(* CoDeSys 2.3 export: BPROOpcion2.EXP *)
(* Libraries: STANDARD.LIB 5.6.98 11:03:02, TcBase.lib 14.5.09 11:14:08, TcBaseMath.lib 27.7.04 11:07:56, TcDrive.lib 25.1.17 09:42:28, TcEtherCAT.lib 30.11.16 19:52:18, TcMath.lib 23.9.04 15:15:30, TcMC2.lib 13.9.17 10:18:38, TcMc2Drive.lib 9.10.17 15:27:28, TcNC.lib 10.10.08 17:55:34, TcSystem.lib 7.6.16 11:01:22, TcTestAndSet.lib 23.2.09 11:50:08, TcUtilities.lib 3.2.16 16:08:58 *)

(* Task configuration *)
TASK Standard (PRIORITY := 0, INTERVAL := T#10ms);
MAIN
END_TASK

(* Global variable list: Global_Variables *)
VAR_GLOBAL
	sCurrentProgram : STRING(20) := 'None';			(* Current Program Loaded or Saved *)

	(* ***** SECURITY ***** *)
	sUsername: STRING := '';
	sPassword : STRING := '';
	sSavePassword : STRING := '';					(* Password Variable for the Save Screen *)
	OldUserLevel : INT := 0;						(* Previous User Level before logging in *)
	CurrentUserLevel : INT :=0;						(* Current User Level*)
	bWrongPassword :BOOL:=FALSE;				(*The password is not correct*)
	bWrongSavePassword :BOOL:=FALSE;				(*The password is not correct*)
	bUserNameHandshake: BOOL := FALSE;			(* Handshake bit to tell panels the User Name Input was received *)
	bPasswordHandshake: BOOL := FALSE;			(* Handshake bit to tell panels the Password Input was received *)
	bSavePasswordHandshake: BOOL := FALSE;		(* Handshake bit to tell panels the Password Input was received *)
	(* SECURITY LEVELS *)
	(* Level 7 - Kays is no longer needed *)
	sUsernameKays : STRING := 'Kays';					(* Username for Kays Engineering *)
	sUsernameKaysLC : STRING := 'kaysengineering';		(* Username for Kays Engineering - Lower Case*)
	sUsernameKaysEngineering : STRING := 'KaysEngineering';		(* Username for Kays Engineering *)
	sPasswordKays : STRING := 'Dehoff';					(* Password for Kays Engineering - Ed's Birthday *)
	(* Level 6 - Maintenance *)
	sUsernameMaint : STRING := 'Maint';					(* Username for Maint *)
	sUsernameMaintLC : STRING := 'maint';				(* Username for maint *)
	sUsernameMaintenance : STRING := 'Maintenance';	(* Username for Maintenance *)
	sUsernameMaintenanceLC : STRING := 'maintenance';	(* Username for maintenance - Lower Case *)
	sPasswordMaint : STRING := 'lazarini';					(* Password for Maintenance - Toggling on the keyboard with the numbers*)
	sPasswordMaintenance : STRING := 'LAZARINI';		(* Password for Maintenance - Toggling on the keyboard with the numbers*)
	(* Level 5 - Supervisor *)
	sUsernameSuper : STRING := 'Super';				(* Username for Super *)
	sUsernameSuperLC : STRING := 'super';				(* Username for super *)
	sUsernameSupervisor : STRING := 'Supervisor';		(* Username for Supervisor *)
	sUsernameSupervisorLC : STRING := 'supervisor';		(* Username for Supervisor  - Lower Case*)
	sPasswordSupervisorUC : STRING := 'ROYALS';		(* Password for Supervisor - Start at 1 and go down then start at 2 and go down keyboard *)
	sPasswordSupervisor : STRING := 'royals';			(* Password for Supervisor - Start at 1 and go down then start at 2 and go down keyboard  - Lower Case*)
	sPasswordSuperUC : STRING := 'ROYALS';		(* Password for Supervisor - Start at 1 and go down then start at 2 and go down keyboard *)
	sPasswordSuper : STRING := 'royals';			(* Password for Supervisor - Start at 1 and go down then start at 2 and go down keyboard  - Lower Case*)

	(* Faulting Variables *)
	bMachineFault: BOOL := FALSE; 					(* Machine Fault Indicator *)
	bMachineWarning: BOOL := FALSE; 				(* Machine Warning Indicator *)
	nFaultArrayIndex : UDINT := 1;
	nWarningArrayIndex : UDINT := 1;
	nModeError : ModeErrors := Er_NoModeError;		(* Errors for different functions *)
	bCoolantTempWarning : BOOL := FALSE;
	bCoolantTempFault : BOOL := FALSE;
	fbCommonFautlResetTON: TON;				(* Trigger of Common Button to Reset Faults *)
	bAFaultResetInternal : BOOL := FALSE;			(* Side A Internal Fault Reset. Triggered by VFD's Ready *)
	bBFaultResetInternal : BOOL := FALSE;			(* Side B Internal Fault Reset. Triggered by VFD's Ready *)
	nActiveFaults: ARRAY[1..4] OF DWORD := 4(0);
	nActiveWarnings: ARRAY[1..4] OF DWORD := 4(0);
	nFaultState: UDINT := 0;
	arrFaultHistory : ARRAY[1..80] OF STRING (52) := 80(''); (* Fault History array *)
	(* Helper Bits *)
	nSetupErrorID: INT :=0;							(* Setup Mode Error Occurred *)
	bLoadSideNotSelected : BOOL := FALSE;
	bTransferError: BOOL := FALSE;					(* An Error Occurred with the Transfer Cycle *)
	nTransferErrorID: INT := 0;						(* Transfer Error ID *)
	sTransferErrorText : STRING := '';				(* Transfer Error Text *)
	(* Parts Tracking *)
	bSideADrilledParts: BOOL := FALSE;				(* Tracking Bit - Side A Completed Drilled parts *)
	bSideBDrilledParts: BOOL := FALSE;				(* Tracking Bit - Side B Completed Drilled parts *)
	fbCoolantLevelDelayTOF: TOF;					(* Delay of the Lowe level switch *)

	(* Status Variables *)
	bMachineMode: BOOL := FALSE;				(* FALSE-->Manual, TRUE-->Automatic *)
	bSetup: BOOL := FALSE;						(* At least one Side in Setup Mode *)
	bSetupA: BOOL := FALSE;						(* In Setup Mode Side A *)
	bSetupB: BOOL := FALSE;						(* In Setup Mode Side B*)
	bInCycle: BOOL := FALSE;						(* In Cycle Flag *)

	(* Cycle Variables *)
	nCycleTimeMinutes : UDINT := 0;
	nCycleTimeSeconds : UDINT := 0;
	nAutoModeState: AutoModeStates := AM_NotInCycle;	(* Counter for Auto Mode State *)
	nAutoCycleStep : AutoCycleStates := AC_Init;		(* Counter for Auto Cycle State *)
	nAC_UnclampStep: INT := 0;					(* Counter for the AC Unclamp Step*)
	bUnloadSideClearOfParts: BOOL :=FALSE;		(* All Unload Side Proxes are off *)
	nCellRunoutCounter: UINT:=0;					(* Counter to keep track of transfer cycles durring Cell Runout *)

	bAutoClampAStart: BOOL := FALSE;				(* Automatic cycle Side A Clamp Parts Tailstock Input *)
	bAutoClampADone: BOOL := FALSE;				(* Automatic cycle Side A Clamp Parts Tailstock Done Output *)
	bAutoClampBStart: BOOL := FALSE;				(* Automatic cycle Side B Clamp PartsTailstock Input *)
	bAutoClampBDone: BOOL := FALSE;				(* Automatic cycle Side B Clamp Parts Tailstock Done Output *)
	bAutoUnclampAStart: BOOL := FALSE;			(* Automatic Side A Unclamp Parts Tailstock Input *)
	bAutoUnclampADone: BOOL := FALSE;			(* Automatic cycle Side A Unclamp Parts Tailstock Done Output *)
	bAutoUnclampBStart: BOOL := FALSE;			(* Automatic Side B Unclamp Parts Tailstock Input *)
	bAutoUnclampBDone: BOOL := FALSE;			(* Automatic cycle Side B Unclamp Parts Tailstock Done Output *)
	bLoadPartsConfirmed: BOOL := FALSE;			(* Operator Confirmed Load Parts In Cycle *)
	bUnloadPartsConfirmed: BOOL := FALSE;			(* Operator Confirmed Unload Parts In Cycle *)
	bAutoTransferPartsToDrill: BOOL := FALSE;		(*Auto Trigger the Transfer to Raise and move parts to Drill Postion*)
	bAutoTransferDownAndLoad : BOOL := FALSE;	(*Auto Trigger the Transfer to lower and move Load Postion*)
	fbProx516TON: TON;							(* Delay of the Transfer Carriage Up Prox *)
	fbProx517TON: TON;							(* Delay of the Transfer Carriage Down Prox *)
	bAutoUpDelayWhileUnclamp: BOOL := FALSE;	(* Auto Helper bit to turn off the up Solenoid when the Unclamp is firing*)

	(*	SERVO VARIABLES *)
	bMCResetRequest: BOOL := FALSE;				(* Request a reset of the NC Axis *)
	bZWADriveResetRequest : BOOL := FALSE;		(* A Side ZW Drive Reset Request *)
	bZBDriveResetRequest : BOOL := FALSE;			(* B Side ZW Drive Reset Request *)
	bZWBDriveResetRequest : BOOL := FALSE;		(* B Side ZW Drive Reset Request *)
	bUDriveResetRequest : BOOL := FALSE;			(* U Axis Drive Reset Request *)
	DriveZAWAdinputs AT %I*: INT;

(* ZA AXIS *)
	stZAAxis: AXIS_REF;
	nZAAxisDiagNumber AT %I*: UDINT := 0;
	nServoZAThrust AT %I* : INT :=0;
	fbZAAxisStop: MC_Stop;
	bZAStop: BOOL := FALSE;
	bZAMCResetRequest: BOOL := FALSE;			(* Request a reset of the NC Axis *)
	fbZAAxisMCReset: MC_Reset;
	fbZAAxisDriveReset : FB_SoEReset;

	bZAAxisEnable: BOOL;
	fbZAAxisPower: MC_Power;
	fbZAAxisMove: MC_MoveAbsolute;
	fbZAAxisSetZero: MC_Home;
	bZAAxisPower: BOOL := FALSE;
	bZAAxisHome: BOOL := FALSE;
	bZAAxisMove: BOOL := FALSE;
	bZAAxisSetZero: BOOL := FALSE;
	fZAMoveVelocity : LREAL := 25.0;
	fZAMovePosition : LREAL := 0.0;
	bZADeCtrlEnable: BOOL := FALSE;				(* Enable for the FB to move off of the Overtravel *)

(* WA AXIS*)
	stWAAxis: AXIS_REF;							(* A Side Tailstock Axis cyclic Interface *)
	nWAAxisDiagNumber AT %I*: UDINT := 0;
	nWAAxisThrust AT %I* : INT :=0;
	fbWAAxisStop: MC_Stop;
	bWAStop: BOOL := FALSE;
	bWAMCResetRequest: BOOL := FALSE;			(* Request a reset of the WA NC Axis *)
	fbWAAxisMCReset: MC_Reset;
	fbWAAxisDriveReset : FB_SoEReset;
	nWATorqeLimitValue AT %Q* : INT := 1000;
	fbWAAxisHome: MC_Home;
	bWAAxisHome: BOOL := FALSE;					(*Trigger the home of WA while homing Automation*)

	DriveZBWBdinputs AT %I*: INT;
(* ZB AXIS *)
	stZBAxis: AXIS_REF;
	nZBAxisDiagNumber AT %I*: UDINT := 0;
	nServoZBThrust AT %I* : INT :=0;
	fbZBAxisStop: MC_Stop;
	bZBStop: BOOL := FALSE;
	bZBMCResetRequest: BOOL := FALSE;			(* Request a reset of the ZA NC Axis *)
	fbZBAxisMCReset: MC_Reset;
	fbZBAxisDriveReset : FB_SoEReset;

	bZBAxisEnable: BOOL;
	fbZBAxisPower: MC_Power;
	fbZBAxisMove: MC_MoveAbsolute;
	fbZBAxisSetZero: MC_Home;
	bZBAxisPower: BOOL := FALSE;
	bZBAxisMove: BOOL := FALSE;
	bZBAxisSetZero: BOOL := FALSE;
	fZBMoveVelocity : LREAL := 25.0;
	fZBMovePosition : LREAL := 0.0;
	bZBDeCtrlEnable: BOOL := FALSE;				(* Enable for the FB to move off of the Overtravel *)

(* WB AXIS *)
	stWBAxis: AXIS_REF;							(* Transfer Axis cyclic Interface *)
	nWBAxisDiagNumber AT %I*: UDINT := 0;
	nWBAxisThrust AT %I* : INT :=0;
	fbWBAxisStop: MC_Stop;
	bWBStop: BOOL := FALSE;
	bWBMCResetRequest: BOOL := FALSE;			(* Request a reset of theWB  NC Axis *)
	fbWBAxisMCReset : MC_Reset;
	fbWBAxisDriveReset : FB_SoEReset;
	nWBTorqeLimitValue AT %Q* : INT  := 1000;
	fbHomeWB: MC_Home;
	bWBAxisHome: BOOL := FALSE;					(*Trigger the home of WB while homing Automation*)

	DriveUdinputs AT %I*: INT;
(* U AXIS 		Also Called X Axis on Screens *)
	stUAxis: AXIS_REF;							(* Transfer Axis cyclic Interface *)
	nUAxisDiagNumber AT %I*: UDINT := 0;
	nUAxisThrust AT %I* : INT :=0;
	fbUAxisStop: MC_Stop;
	bUStop: BOOL := FALSE;
	bUMCResetRequest: BOOL := FALSE;			(* Request a reset of the U NC Axis *)
	fbUAxisMCReset : MC_Reset;
	fbUAxisDriveReset : FB_SoEReset;
	fbTransferAxisHome: MC_Home;
	bUAxisHome: BOOL := FALSE;					(*Trigger the home of U Axis while homing Automation*)
	fTransferMoveVelo : LREAL := 0.0;				(* Velocity to pass to the U Axis Move FB *)

(* MPG Axis Definitions *)
	stAxisMPG_A : Axis_REF;						(* Side A MPG Axis Cyclic Interface *)
	fbMPGAAxisMCReset: MC_Reset;
	stAxisMPG_B : Axis_REF;						(* Side A MPG Axis Cyclic Interface *)
	fbMPGBAxisMCReset: MC_Reset;
	bMPGA_MCResetRequest: BOOL := FALSE;		(* Axis Reset of the MPGA Axis *)
	bMPGB_MCResetRequest: BOOL := FALSE;		(* Axis Reset of the MPGB Axis *)
	bMPGAOn: BOOL := FALSE;						(* MPG A has an axis selected *)
	bMPGBOn: BOOL := FALSE;						(* MPG B has an axis selected *)

(* VFD Control Variables - EtherCAT Emerson *)
	fbGetAMS: FB_GetAxisAmsAddr;
	fbVFD_A1: FB_EtherCAT_Emerson;
	bVFD_A1DataValid AT %I*: BOOL;				(* Must Asign to VFD WcStateIn in System Manager*)
	fbVFD_A2: FB_EtherCAT_Emerson;
	bVFD_A2DataValid AT %I*: BOOL;				(* Must Asign to VFD WcStateIn in System Manager*)
	fbVFD_A3: FB_EtherCAT_Emerson;
	bVFD_A3DataValid AT %I*: BOOL;				(* Must Asign to VFD WcStateIn in System Manager*)
	fbVFD_B1: FB_EtherCAT_Emerson;
	bVFD_B1DataValid AT %I*: BOOL;				(* Must Asign to VFD WcStateIn in System Manager*)
	fbVFD_B2: FB_EtherCAT_Emerson;
	bVFD_B2DataValid AT %I*: BOOL;				(* Must Asign to VFD WcStateIn in System Manager*)
	fbVFD_B3: FB_EtherCAT_Emerson;
	bVFD_B3DataValid AT %I*: BOOL;				(* Must Asign to VFD WcStateIn in System Manager*)
	bVFD_ARun: BOOL := FALSE;
	bVFD_BRun: BOOL := FALSE;
	bVFDControlDirection: BOOL := FALSE;
	fVFDControlRatio: LREAL := 1.0;
	bVFD_A1UpToSpeed: BOOL := FALSE;
	bVFD_A1Error: BOOL := FALSE;
	nVFD_A1ErrorID: UDINT := 0;
	stVFD_A1DriveInfo: Ke_VFDInfo;
	bVFD_A2UpToSpeed: BOOL := FALSE;
	bVFD_A2Error: BOOL := FALSE;
	nVFD_A2ErrorID: UDINT := 0;
	stVFD_A2DriveInfo: Ke_VFDInfo;
	bVFD_A3UpToSpeed: BOOL := FALSE;
	bVFD_A3Error: BOOL := FALSE;
	nVFD_A3ErrorID: UDINT := 0;
	stVFD_A3DriveInfo: Ke_VFDInfo;
	bVFD_B1UpToSpeed: BOOL := FALSE;
	bVFD_B1Error: BOOL := FALSE;
	nVFD_B1ErrorID: UDINT := 0;
	stVFD_B1DriveInfo: Ke_VFDInfo;
	bVFD_B2UpToSpeed: BOOL := FALSE;
	bVFD_B2Error: BOOL := FALSE;
	nVFD_B2ErrorID: UDINT := 0;
	stVFD_B2DriveInfo: Ke_VFDInfo;
	bVFD_B3UpToSpeed: BOOL := FALSE;
	bVFD_B3Error: BOOL := FALSE;
	nVFD_B3ErrorID: UDINT := 0;
	stVFD_B3DriveInfo: Ke_VFDInfo;
	nVFD_A1Addr AT %I*: UINT := 0;						(*Spindle#A1 VFD Slave Addres Input Variable*)
	nVFD_A2Addr AT %I*: UINT := 0;						(*Spindle#A1 VFD Slave Addres Input Variable*)
	nVFD_A3Addr AT %I*: UINT := 0;						(*Spindle#A1 VFD Slave Addres Input Variable*)
	nVFD_B1Addr AT %I*: UINT := 0;						(*Spindle#A1 VFD Slave Addres Input Variable*)
	nVFD_B2Addr AT %I*: UINT := 0;						(*Spindle#A1 VFD Slave Addres Input Variable*)
	nVFD_B3Addr AT %I*: UINT := 0;						(*Spindle#A1 VFD Slave Addres Input Variable*)


(* Solenoid Auto Control Variables *)
	bAutoLower: BOOL := FALSE;						(* Auto Lower Transfer Carrier Cylinder*)
	bAutoRaise: BOOL := FALSE;						(* Auto Raise Transfer Carrier Cylinder*)
	bAAutoOpenCollet: BOOL := FALSE;					(* Auto Control to Open the Collets on Side A*)
	bAAutoCloseCollet: BOOL := FALSE;					(* Auto Control to Close the Collets on Side A*)
	bBAutoOpenCollet: BOOL := FALSE;					(* Auto Control to Open the Collets on Side B*)
	bBAutoCloseCollet: BOOL := FALSE;					(* Auto Control to Close the Collets on Side B*)
	bAAutoEjectorsAdvance: BOOL := FALSE;				(* Auto Control to Advance the Ejectors on Side A *)
	bAAutoEjectorsRetract: BOOL := FALSE;				(* Auto Control to Retract the Ejectors on Side A *)
	bBAutoEjectorsAdvance: BOOL := FALSE;				(* Auto Control to Advance the Ejectors on Side A *)
	bBAutoEjectorsRetract: BOOL := FALSE;				(* Auto Control to Retract the Ejectors on Side A *)

	bWandUAxisHomed: BOOL := FALSE;				(* The W and U Axis are Homed*)

	nAEjectorAdvancedState: USINT := 0;
	nAEjectorRetractedState: USINT := 0;
	nBEjectorAdvancedState: USINT := 0;
	nBEjectorRetractedState: USINT := 0;

(* Tailstock Variables *)
	Side_A_Fixture: FB_FixtureControl;					(*Side A Tailstock Control FB*)
	Side_B_Fixture: FB_FixtureControl;					(*Side B Tailstock Control FB*)
	fWAxisFastVelocity: LREAL := 0.0;					(*WA and WB Axis Velocity to Feed to Tailstock FB*)
	fWAxisClampVelocity: LREAL := 0.0;					(*WA and WB Axis Clamp Velocity to Feed to Tailstock FB*)

END_VAR

VAR_GLOBAL PERSISTENT

	sSerialNumber : STRING(20) := 'DH-2062';				(* This holds the serial number of the machine *)
	sKaysJobNumber  : STRING(20) := '6216';				(* This holds the Kayse Engineering Job number of the machine *)
	sModelNumber : STRING(20) := '6-Spindle Special';		(* This variable holds the model of the machine *)
	sCustomerName : STRING(20) := 'ARBOMEX';			(* This variable holds the customers name *)
	nMachineNumber : UDINT := 7;						(* The Machine Number designates what number the machines were delivered in for this series of special machines *)
	sProductionDate : STRING(10) := '01/2016';			(* This variable holds the date of production and should match that of the machine tags *)

	sLoadSideSet : STRING(30) :='None';					(* Holds the side that is currently set as Infeed *)
	bSideAEnabled : BOOL := TRUE;					(* Enable of Machine Side A *)
	bSideBEnabled : BOOL := TRUE;					(* Enable of Machine Side B *)
	fFlowMonitorMax : LREAL := 0;						(* Max set in program *)

	nMaxCycles : UDINT := 0;							(* Max Cycles set in program *)
	nCyclesComplete : UDINT := 0;						(* Completed # of Cycles since Reset *)

	sLastLoadedPartProgramName : STRING(25) := 'None';	(* Stores the Name of the Last Part Program Loaded *)
	nMotorNominalRPM : UDINT := 3460;

	(* Tailstock Variables *)
	nWAAxisThrustMax: UDINT := 40;					(* Tailstock WA Axis Max Thrust *)
	nWBAxisThrustMax: UDINT := 40;					(* Tailstock WB Axis Max Thrust *)
	fWAAxisHomeOffset : LREAL := 0.0;					(* A Tailstock WA Axis Offset Durring Homing *)
	fWBAxisHomeOffset : LREAL := 0.0;					(* B Tailstock WB Axis Offset Durring Homing *)
	fWAxisMoveOffBushing : LREAL := 0.0;				(* Amount to Back W Axis' off of Bushing After Drill *)
	nTailstockClampingTorqueLimit : INT := 15;			(* % Torque Limit for W Axis During Clamp for Drilling *)
	fTailstockVelocity : LREAL := 60.0;					(* Velocity of the W Axis for normal moves*)
	fTailstockClampVelocity : LREAL := 30.0;				(* Velocity of the W Axis for the move to Clamp position *)
	(* Transfer Position and Speeds - U Axis *)
	fUAxisLoadSidePosition: LREAL := 0.0;				(* Transfer Axis Servo Load Position *)
	fUAxisUnloadSidePosition: LREAL := 0.0;				(* Transfer Axis Servo Unload Position *)
	fUAxisVelocity: LREAL := 0.0;						(* Transfer Axis Servo Move Speed *)
	nUAxisThrustMax : UDINT :=100;						(* Max Thrust Set in secret screen *)

END_VAR

(* Global variable list: Inputs *)
VAR_GLOBAL
(* Rack 1 Slot 1 -EL1809 *)
	bPB1AConfirm AT %I* : BOOL := FALSE;				(* A -Load/Unload Confirm *)
	bPB2ACycleStart AT %I* : BOOL := FALSE;			(* A -Cycle Start PB *)
	bPB3ACycleCommon AT %I* : BOOL := FALSE;		(* A -Cycle Common/Reset PB *)
	bPB4ADrillReturn AT %I* : BOOL := FALSE;			(* A -Drill Return PB *)
	bPB1BConfirm AT %I* : BOOL := FALSE;				(* B -Load/Unload Confirm *)
	bPB2BCycleStart AT %I* : BOOL := FALSE;			(* B -Cycle Start PB *)
	bPB3BCycleCommon AT %I* : BOOL := FALSE;		(* B -Cycle Common/Reset PB *)
	bPB4BDrillReturn AT %I* : BOOL := FALSE;			(* B -Drill Return PB *)
	bChipConveyorVFDFault AT %I* : BOOL := FALSE;		(*  Chip Conveyor VFD Fault feedback *)
	(*Spare*)
	bCleanTankLevel AT %I* : BOOL := FALSE;			(* FS1 *)
	bCoolantTankOverflow AT %I* : BOOL := FALSE;		(* FS2 *)
	bFilter1Dirty AT %I* : BOOL := FALSE;					(* DPS1 *)
	bFilter2Dirty AT %I* : BOOL := FALSE;					(* DPS2 *)
	bFilter3Dirty AT %I* : BOOL := FALSE;					(* DPS3 *)
	bFilter4Dirty AT %I* : BOOL := FALSE;					(* DPS4 *)

(* Rack 1 Slot 2 - EL1809 *)
	bACoolantPressure AT %I* : BOOL := FALSE;			(* PS1 *)
	bBCoolantPressure AT %I* : BOOL := FALSE;			(* PS2 *)
	bLubeLevel AT %I* : BOOL := FALSE;					(* FS3 *)
	bLubePressure AT %I* : BOOL := FALSE;				(* PS3 *)
	bHydraulicSystemLevel AT %I* : BOOL := FALSE;		(* FS4 *)
	bHydraulicSystemPressure AT %I* : BOOL := FALSE;	(* PS4 *)
	bHydraulicTemperature AT %I* : BOOL := FALSE;		(* TS1 *)
	(*Spare*)
	bPneumaticSystemPressure AT %I* : BOOL := FALSE;	(* PS5 *)
	(*Spare*)
	bMCC_SConfirm AT %I* : BOOL := FALSE;			 	(* Servo Master Control Relay Active	*)
	(*Spare*)
	(*Spare*)
	(*Spare*)
	(*Spare*)
	bMCR AT %I* : BOOL := FALSE; 						(* Master Control Relay Active	*)

(* Rack 1 Slot 3 - EL1809 *)
	(* All Spares *)

(* Rack 1 Slot 3 - EL3311 *)
	nCoolantTemp AT %I* : INT := 0;

(* Rack 1 Slot 7 - EL3152  *)
	nSpindleTachA1 AT %I* : INT := 0;
	nCoolantFlowA1 AT %I* : INT :=0;

(* Rack 1 Slot 8 - EL3152 *)
	nSpindleTachA2 AT %I* : INT := 0;
	nCoolantFlowA2 AT %I* : INT :=0;

(* Rack 1 Slot 9 - EL3152 *)
	nSpindleTachA3 AT %I* : INT := 0;
	nCoolantFlowA3 AT %I* : INT :=0;

(* Rack 1 Slot 11 - EL3152  *)
	nSpindleTachB1 AT %I* : INT := 0;
	nCoolantFlowB1 AT %I* : INT :=0;

(* Rack 1 Slot 12 - EL3152 *)
	nSpindleTachB2 AT %I* : INT := 0;
	nCoolantFlowB2 AT %I* : INT :=0;

(* Rack 1 Slot 13 - EL3152 *)
	nSpindleTachB3 AT %I* : INT := 0;
	nCoolantFlowB3 AT %I* : INT :=0;

(* Rack 1 Slot 15 - EL1008 *)
	bZAAxisSelected AT %I* : BOOL := FALSE;		(* MPG Side A Z Selected *)
	bARate1X AT %I* : BOOL := FALSE;
	bARate10X AT %I* : BOOL := FALSE;
	bARate100X AT %I* : BOOL := FALSE;
	bWAAxisSelected AT %I* : BOOL := FALSE;
	bXAAxisSelected AT %I* : BOOL := FALSE;
	bYAAxisSelected AT %I* : BOOL := FALSE;
	(*SPARE*)

(* Rack 2 Slot 3 - EL1008 *)
	bZBAxisSelected AT %I* : BOOL := FALSE;		(* MPG Side A Z Selected *)
	bBRate1X AT %I* : BOOL := FALSE;
	bBRate10X AT %I* : BOOL := FALSE;
	bBRate100X AT %I* : BOOL := FALSE;
	bWBAxisSelected AT %I* : BOOL := FALSE;
	bXBAxisSelected AT %I* : BOOL := FALSE;
	bYBAxisSelected AT %I* : BOOL := FALSE;
	(*SPARE*)

(* Rack 2 Slot 4 - EL1008 *)
	bHighPressureMotorRunning AT %I* : BOOL := FALSE;
	bTransferPumpMotorRunning AT %I* : BOOL := FALSE;
	bChipConveyorMotorRunning AT %I* : BOOL := FALSE;
	bHydraulicPowerUnitRunning AT %I* : BOOL := FALSE;
	bMCC_V AT %I* : BOOL := FALSE;					(* Spindle Drives Power Enabled Feedback *)
	(*SPARE*)
	(*SPARE*)
	(*SPARE*)

(* Rack 2 Slot 5 - EL1008 *)
	(* All Spares *)

(* Rack 3 - EP1008 *)
	bProx310 AT %I* : BOOL := FALSE;			(* A Side - Sliding Door Closed *)
	bProx311 AT %I* : BOOL := FALSE;			(* B Side - Sliding Door Closed *)
	bProx312 AT %I* : BOOL := FALSE;			(* A Side - Fixture Door Closed *)
	bProx313 AT %I* : BOOL := FALSE;			(* B Side - Fixture Door Closed *)
	(*SPARE*)
	(*SPARE*)
	(*SPARE*)
	(*SPARE*)
	bRack3Comm AT %I* : BOOL := FALSE;		(* Ethercat Comm Status to Rack 3 *)

(* Rack 4 - EP1008 *)
	(* A Side Conveyor PROX Indicators *)
	bProx410 AT %I* : BOOL := FALSE;			(* A -Spindle 1 *)
	bProx411 AT %I* : BOOL := FALSE;			(* A -Spindle 2 *)
	bProx412 AT %I* : BOOL := FALSE;			(* A -Spindle 3 *)
	bProx413 AT %I* : BOOL := FALSE;			(* B -Spindle 1 *)
	bProx414 AT %I* : BOOL := FALSE;			(* B -Spindle 2 *)
	bProx415 AT %I* : BOOL := FALSE;			(* B -Spindle 3 *)
	(*SPARE*)
	(*SPARE*)
	bRack4Comm AT %I* : BOOL := FALSE;		(* Ethercat Comm Status to Rack 4 *)

(* Rack 5 - EP1008 *)
	(* B Side Conveyor PROX Indicators *)
	bProx510 AT %I* : BOOL := FALSE;			(* A -Spindle 1 *)
	bProx511 AT %I* : BOOL := FALSE;			(* A -Spindle 2 *)
	bProx512 AT %I* : BOOL := FALSE;			(* A -Spindle 3 *)
	bProx513 AT %I* : BOOL := FALSE;			(* B -Spindle 1 *)
	bProx514 AT %I* : BOOL := FALSE;			(* B -Spindle 2 *)
	bProx515 AT %I* : BOOL := FALSE;			(* B -Spindle 3 *)
	bProx516 AT %I* : BOOL := FALSE;			(* Carrier Up *)
	bProx517 AT %I* : BOOL := FALSE;			(* Carrier Down *)
	bRack5Comm AT %I* : BOOL := FALSE;		(* Ethercat Comm Status to Rack 5 *)

(* Rack 6 - EP1008 *)
	(* A Side Ejector PROX Indicators *)
	bProx610 AT %I* : BOOL := FALSE;			(* A Part Ejector #1 Retracted *)
	bProx611 AT %I* : BOOL := FALSE;			(* A Part Ejector #2 Retracted *)
	bProx612 AT %I* : BOOL := FALSE;			(* A Part Ejector #3 Retracted *)
	bProx613 AT %I* : BOOL := FALSE;			(* A Part Ejector #1 Advanced *)
	bProx614 AT %I* : BOOL := FALSE;			(* A Part Ejector #2 Advanced *)
	bProx615 AT %I* : BOOL := FALSE;			(* A Part Ejector #3 Advanced *)
	bPS616 AT %I* : BOOL := FALSE;			(* A Collets Unclamp Pressure Switch *)
	bPS617 AT %I* : BOOL := FALSE;			(* A Collets Clamp Pressure Switch *)
	bRack6Comm AT %I* : BOOL := FALSE;		(* Ethercat Comm Status to Rack 6 *)

(* Rack 7 - EP1008 *)
	(* B Side Ejector PROX Indicators *)
	bProx720 AT %I* : BOOL := FALSE;			(* B Part Ejector #1 Retracted *)
	bProx721 AT %I* : BOOL := FALSE;			(* B Part Ejector #2 Retracted *)
	bProx722 AT %I* : BOOL := FALSE;			(* B Part Ejector #3 Retracted *)
	bProx723 AT %I* : BOOL := FALSE;			(* B Part Ejector #1 Advanced *)
	bProx724 AT %I* : BOOL := FALSE;			(* B Part Ejector #2 Advanced *)
	bProx725 AT %I* : BOOL := FALSE;			(* B Part Ejector #3 Advanced *)
	bPS726 AT %I* : BOOL := FALSE;			(* B Collets Unclamp Pressure Switch *)
	bPS727 AT %I* : BOOL := FALSE;			(* B Collets Clamp Pressure Switch *)
	bRack7Comm AT %I* : BOOL := FALSE;		(* Ethercat Comm Status to Rack 7 *)

END_VAR

(* Global variable list: Network_Variables *)
VAR_GLOBAL
(* Subscribe to Panel A *)
	stReceivePanelA AT %I* : ST_PANEL_SEND;		(* Structure of Push Buttonas and Inputs from Panel A *)
	nReceivePanelAQuality AT %I* : UINT :=0;			(* Good Quality is 0 when receiving data from Panel A *)
	nReceivePanelACycleIndex AT %I* : UINT :=0;		(* Cycle Index Continures to change while receiving data from Panel A *)
	(* Requests by Panel A for the CX to place network variables on the network *)
	nRequestPA AT %I* : WORD := 0;

(* Subscribe to Panel B *)
	stReceivePanelB AT %I* : ST_PANEL_SEND;		(* Structure of Push Buttonas and Inputs from Panel B *)
	nReceivePanelBQuality AT %I* : UINT :=0;			(* Good Quality is 0 when receiving data from Panel B *)
	nReceivePanelBCycleIndex AT %I* : UINT :=0;		(* Cycle Index Continures to change while receiving data from Panel B *)
	(* Requests by Panel A for the CX to place network variables on the network *)
	nRequestPB AT %I* : WORD := 0;

(* Publish Variables *)
	(* Structure for the CX Publish Variable 1 *)
	stCXPublish1 AT %Q* : ST_CX_Publish1;
	(* Array of String Variables for Machine Information -  Only required at power up of CP2612's *)
	arrMachineInfo AT %Q* : ARRAY[1..20] OF STRING(30) := 20('');
	(* Structure to display of the Part Program - only sent when on the Part Program screen *)
	stPartProgramSend AT %Q* : ST_PARTPROGRAM;
	(* Structure of the VFD Information *)

(* Variable Controol  - A value of 1 disables publishing, 0 enables *)
	nPubFrameState AT %I* : UINT :=0;				(* Frame State of the Published Network Variable - 1=not sent, 2=oversized Error *)
	nVarCtrlMachineInfo AT %Q* : UINT := 1;			(*Variable Control for the Text Array for Main Screen*)
	nVarCtrlAutoDisplays AT %Q* : UINT :=1;			(* Variable Control for the Auto Display Net Variables *)
	nVarCtrlFaultMessages AT %Q* : UINT := 1;		(* Variable Control for the Fault Messages Net Variables *)
	nVarCtrlPanelReceive AT %Q* : UINT := 0;			(* Variable Control for Panel Information - Always 0 *)
	nVarCtrlPartProgramSend AT %Q* : UINT :=0;		(* Variable Control for Part Program Send *)
	nVarCtrlDemo AT %Q* : UINT := 1;				(* Variable Control for the Demo Net Variables *)

(*Demo Variables*)
	stPB AT %I* : ST_Demo_PBs;					(* Define a structure of the push buttons to be recieved from the panel A *)
	stPBB AT %I* : ST_Demo_PBs;					(* Define a structure of the push buttons to be recieved from the panel B*)
	stLT AT %Q* : ST_Demo_Indicators;				(* Define a structure of the Lights to be sent to the panel *)

END_VAR

(* Global variable list: Outputs *)
VAR_GLOBAL

(* Rack 1 Slot 5 EL2809 *)
	bAServoEnable AT %Q* : BOOL := FALSE;			(* A side Servo Hard Enable Relay *)
	bBServoEnable AT %Q* : BOOL := FALSE;			(* B side Servo Hard Enable Relay *)
	bUServoEnable AT %Q* : BOOL := FALSE;			(* Transfer Servo Hard Enable Relay *)
	bMCC_S AT %Q* : BOOL := FALSE;					(* Servo Power Delayed Contactor *)
	bWayLubePump AT %Q* : BOOL := FALSE;			(* Way Lube Pump Power *)
	bACoolantSolenoid AT %Q* : BOOL := FALSE;			(* A Side Coolant Solenoid On SOL1 *)
	bBCoolantSolenoid AT %Q* : BOOL := FALSE;			(* B Side Coolant Solenoid On SOL2 *)
	bConveyorFWDReq AT %Q* : BOOL := FALSE;		(* Chip Conveyor Forward Request *)
	bHPCoolantStart_A AT %Q* : BOOL := FALSE;			(* A Side High Pressure Coolant Soft Start SOL 4 *)
	bHPCoolantStart_B AT %Q* : BOOL := FALSE;			(* B Side High Pressure Coolant Soft Start SOL 5 *)
	bTransferDown AT %Q* : BOOL := FALSE;				(* Lower Transfer Solenoid *)
	bTransferUp AT %Q* : BOOL := FALSE;				(* Raise Transfer Solenoid *)
	bATailstockColletUnclamp AT %Q* : BOOL := FALSE;	(* Unclamp Collet Solenoid Side A *)
	bATailstockColletClamp AT %Q* : BOOL := FALSE;		(* Clamp Collet Solenoid Side A *)
	bBTailstockColletUnclamp AT %Q* : BOOL := FALSE;	(* Unclamp Collet Solenoid Side B *)
	bBTailstockColletClamp AT %Q* : BOOL := FALSE;		(* Clamp Collet Solenoid Side B *)

(* Rack 1 Slot 6 EL2809 *)
	bAEjectorsRetract AT %Q* : BOOL := FALSE;			(* Side A Ejectors/Pushers Retract *)
	bAEjectorsAdvance AT %Q* : BOOL := FALSE;			(* Side A Ejectors/Pushers Advance *)
	bBEjectorsRetract AT %Q* : BOOL := FALSE;			(* Side B Ejectors/Pushers Retract *)
	bBEjectorsAdvance AT %Q* : BOOL := FALSE;			(* Side B Ejectors/Pushers Advance *)
	(* SPARE*)
	(* SPARE*)
	(* SPARE*)
	(* SPARE*)
	bChipConveyorFWD AT %Q* : BOOL := FALSE;
	(* SPARE*)
	bLT2 AT %Q* : BOOL := FALSE;						(* Light Tower - Fault *)
	bLT3 AT %Q* : BOOL := FALSE;						(* Light Tower - Idle *)
	bLT4 AT %Q* : BOOL := FALSE;						(* Light Tower -  In Cycle *)
	bLT5 AT %Q* : BOOL := FALSE;						(* Fault Light - Side A *)
	(* SPARE*)
	(* SPARE*)

(* Rack 2 Slot 6 EL2008 *)
	bLT6 AT %Q* : BOOL := FALSE;					(* Fault Light - Side B *)
	bHighPressureMotorOn AT %Q* : BOOL := FALSE;
	bTransferPumpOn AT %Q* : BOOL := FALSE;
	bHydraulicUnitOn AT %Q* : BOOL := FALSE;
	bChipConveyorOn AT %Q* : BOOL := FALSE;
	(* SPARE*)
	(* SPARE*)
	(* SPARE*)

(* Rack 2 Slot 7 EL2008 *)
	bVFD_A_Enable AT %Q* : BOOL := FALSE;
	bVFD_B_Enable AT %Q* : BOOL := FALSE;
	(* SPARE*)
	(* SPARE*)
	(* SPARE*)
	(* SPARE*)
	(* SPARE*)
	(* SPARE*)

END_VAR

(* Global variable list: SCREEN_DISPLAYS *)
VAR_GLOBAL
(* MASTER Layout *)
	nEtherCATMasterState: INT := 0;
	sScreenTitle : STRING(45) := '';
	sCurrentCXProgram : STRING(25) := 'None';		(* Current Program in the CX Processor *)
	bDispPressCycleStart: BOOL := FALSE;			(* Trigger when Cycle Start is necessary to resume operation *)

(* MANUAL Screen *)
	(* Push Buttons *)
	bStartHydraulicPB : BOOL := FALSE;				(* Start the Hydraulic Unit *)
	bStopHydraulicPB : BOOL := FALSE;				(* Start the Hydraulic Unit *)
	bCoolantStartPB : BOOL := FALSE;				(* Start the Coolant System *)
	bCoolantStopPB : BOOL := FALSE;				(* Stop the Coolant System *)
	bEnterSetupPB_A : BOOL := FALSE;				(* Side A Enter Setup Mode *)
	bEnterSetupPB_B : BOOL := FALSE;				(* Side B Enter Setup Mode *)
	bSetZeroPositionPB_A : BOOL := FALSE;			(* Set ZA Azis Position to Zero *)
	bSetZeroPositionPB_B : BOOL := FALSE;			(* Set ZB Azis Position to Zero *)
	bMoveToZeroPositionPB_A : BOOL := FALSE;		(* Move ZA Axis to Zero Positon *)
	bMoveToZeroPositionPB_B : BOOL := FALSE;		(* Move ZB Axis to Zero Positon *)
	bHomeAutomationPB : BOOL := FALSE;			(* Home WA, WB, and X Axis *)

(* AUTO Screen *)
	(* SPINDLE VARIABLES *)
	nSpindleRPM1A: UDINT := 0;
	nSpindleRPM2A: UDINT := 0;
	nSpindleRPM3A: UDINT := 0;
	nSpindleRPM1B: UDINT := 0;
	nSpindleRPM2B: UDINT := 0;
	nSpindleRPM3B: UDINT := 0;
	nSpindleLoad1ADisplay : UDINT := 0;
	nSpindleLoad2ADisplay : UDINT := 0;
	nSpindleLoad3ADisplay : UDINT := 0;
	nSpindleLoad1BDisplay : UDINT := 0;
	nSpindleLoad2BDisplay : UDINT := 0;
	nSpindleLoad3BDisplay : UDINT := 0;
	nSpindleLoadMax : UDINT := 100;
	(* Coolant *)
	fCoolantFlow1ADisplay : LREAL := 0;
	fCoolantFlow1AGraph: LREAL := 0;
	fCoolantFlow2ADisplay : LREAL := 0;
	fCoolantFlow2AGraph: LREAL := 0;
	fCoolantFlow3ADisplay : LREAL := 0;
	fCoolantFlow3AGraph: LREAL := 0;
	fCoolantFlow1BDisplay : LREAL := 0;
	fCoolantFlow1BGraph: LREAL := 0;
	fCoolantFlow2BDisplay : LREAL := 0;
	fCoolantFlow2BGraph: LREAL := 0;
	fCoolantFlow3BDisplay : LREAL := 0;
	fCoolantFlow3BGraph: LREAL := 0;
	fCoolantTempDisplay: LREAL := 0.0;
	fCoolantFlowMinGraph: LREAL := 0.0;
	fCoolantFlowMaxGraph: LREAL := 0.0;

	(* Servo Variables *)
	fZAAxisVelosity : LREAL := 0.0;						(* ZA Axis Velocity/Feedrate *)
	fZBAxisVelosity : LREAL := 0.0;						(* ZB Axis Velocity/Feedrate *)
	nServoAThrustDisplay : UDINT := 0;
	nServoBThrustDisplay : UDINT := 0;
	nServoThrustMax : UDINT := 100;

	(* Cycle Variables *)
	nPartsCompleteTotal : UDINT := 0;
	nPartsCompleteA1 : UDINT := 0;
	nPartsCompleteA2 : UDINT := 0;
	nPartsCompleteA3 : UDINT := 0;
	nPartsCompleteB1 : UDINT := 0;
	nPartsCompleteB2 : UDINT := 0;
	nPartsCompleteB3 : UDINT := 0;

	bCellRunOutRequest : BOOL := FALSE;				(* Cell Runout has been requested *)
	bCellRunOutPB: BOOL := FALSE;

	(* Push Buttons *)
	bEnterManualModePB: BOOL := FALSE;
	bEnterAutoModePB: BOOL := FALSE;
	bResetCycleCounterPB: BOOL := FALSE;
	bFaultResetPB: BOOL := FALSE;
	bResetTotalCountPB: BOOL := FALSE;
	bResetA1CountPB: BOOL := FALSE;
	bResetA2CountPB: BOOL := FALSE;
	bResetA3CountPB: BOOL := FALSE;
	bResetB1CountPB: BOOL := FALSE;
	bResetB2CountPB: BOOL := FALSE;
	bResetB3CountPB: BOOL := FALSE;

	sCurrentPartProgram : STRING(25) := 'None';		(* Current Part Program Loaded*)

(* The Fault Messages is transfered and used as is *)
	arrFaultMessage : ARRAY[1..10] OF STRING (50) := 10('');

(* PART PROGRAM STORAGE VARIABLES *)
	sPartProgramName : STRING(25) := 'None';
	bPartProgramSavePB : BOOL := FALSE;
	bPartProgramLoadPB : BOOL := FALSE;

	fStartFeed : LREAL := 0.0;
	fFinishFeed : LREAL := 0.0;
	fStartDepth : LREAL := 0.0;
	fFinishDepth : LREAL := 0.0;
	fDwellTime : LREAL := 0.0;
	fRetractRate : LREAL := 0.0;
	fDrillTipOffset : LREAL := 0.0;
	fRPMRequest : LREAL := 0.0;
	fToolDiameter : LREAL := 0.0;
	fCoolantPressure : LREAL := 0.0;
	fCoolantFlowMax : LREAL := 0.0;
	fCoolantFlowMin : LREAL := 0.0;

	bSpindleRetractMode : BOOL := FALSE;
	bFaultHistoryFileError : BOOL := FALSE;

	sFileOpError : STRING(30) := '';

	bStartFeedChanged: BOOL := FALSE;			(*Indicates Start Feed changed since program was loaded*)
	bFinishFeedChanged: BOOL := FALSE;			(*Indicates changed since program was loaded*)
	bStartDepthChanged: BOOL := FALSE;			(*Indicates changed since program was loaded*)
	bFinishDepthChanged: BOOL := FALSE;			(*Indicates changed since program was loaded*)
	bDwellTimeChanged: BOOL := FALSE;			(*Indicates changed since program was loaded*)
	bRetractRateChanged: BOOL := FALSE;			(*Indicates changed since program was loaded*)
	bDrillTipOffsetChanged: BOOL := FALSE;			(*Indicates changed since program was loaded*)
	bRPMRequestChanged: BOOL := FALSE;			(*Indicates changed since program was loaded*)
	bSpindleRetractChanged: BOOL := FALSE;		(*Indicates changed since program was loaded*)
	bToolDiameterChanged: BOOL := FALSE;			(*Indicates changed since program was loaded*)
	bSpindleLoadMaxChanged: BOOL := FALSE;		(*Indicates changed since program was loaded*)
	bServoThrustMaxChanged: BOOL := FALSE;		(*Indicates changed since program was loaded*)
	bCoolantFlowMaxChanged: BOOL := FALSE;		(*Indicates changed since program was loaded*)
	bCoolantFlowMinChanged: BOOL := FALSE;		(*Indicates changed since program was loaded*)
	bMaxCyclesChanged: BOOL := FALSE;			(*Indicates changed since program was loaded*)

(* TRANSFER Variables *)
	(* Displays *)
	bTransferUpPX : BOOL := FALSE;				(* Transfer Up Indicator *)
	bTransferDownPX : BOOL := FALSE;				(* Transfer Down Indicator *)
	bTransferUpSOL: BOOL :=FALSE;				(* Transfer Up Solenoid *)
	bTransferDownSOL : BOOL := FALSE;			(* Transfer Down Solenoid *)

	(* Operators*)
	bTransferUpPB : BOOL := FALSE;				(* Transfer Up Push Button *)
	bTransferDownPB : BOOL := FALSE;				(* Transfer Down Push Button *)
	bHomeUAxisPB : BOOL := FALSE;				(* Home U Axis Push Button *)
	bMoveUtoLoadPB : BOOL := FALSE;				(* Move U Axis to Load Position Push Button *)
	bMoveUtoUnloadPB : BOOL := FALSE;			(* Move U Axis to Unload Position Push Button *)
	bTransferAtLoadIndicator : BOOL := FALSE;		(* Indicator that Transfer At the Load Position *)
	bTransferAtUnloadIndicator : BOOL := FALSE;		(* Indicator that Transfer At the Unload Position *)

(* FIXTURE/TAILSTOCK Variables *)
	fWAxisTransferPosition : LREAL := 0.0;			(* Tailstock W Axis Position During Transfer *)
	fWAxisDrillPosition : LREAL := 0.0;				(* Tailstock W Axis Position During Drill *)

	(* A Side *)
	bAEjectorOvertravelError : BOOL := FALSE;		(* One of the Ejectors has overtraveled *)
	(* Push Buttons - Operators *)
	bWAAxisHomePB : BOOL := FALSE;				(* Tailstock WA Axis Home *)
	bWAAxisAdvancePB : BOOL := FALSE;			(* Tailstock WA Axis Advance Postion *)
	bWAAxisRetractPB : BOOL := FALSE;				(* Tailstock WA Axis Retract Postion *)
	bAColletClosePB : BOOL := FALSE;				(* Tailstock A Close Collets *)
	bAColletOpenPB : BOOL := FALSE;				(* Tailstock A Open Collets *)
	bAEjectorsAdvancePB : BOOL := FALSE;			(* Tailstock A Advance Ejectors *)
	bAEjectorsRetractPB : BOOL := FALSE;			(* Tailstock A Retract Ejectors *)

	(* B Side *)
	bBEjectorOvertravelError : BOOL := FALSE;		(* One of the Ejectors has overtraveled *)
	(* Push Buttons - Operators *)
	bWBAxisHomePB : BOOL := FALSE;				(* Tailstock WB Axis Home *)
	bWBAxisAdvancePB : BOOL := FALSE;			(* Tailstock WB Axis Advance Postion *)
	bWBAxisRetractPB : BOOL := FALSE;				(* Tailstock WB Axis Retract Postion *)
	bBColletClosePB : BOOL := FALSE;				(* Tailstock B Close Collets *)
	bBColletOpenPB : BOOL := FALSE;				(* Tailstock B Open Collets *)
	bBEjectorsAdvancePB : BOOL := FALSE;			(* Tailstock B Advance Ejectors *)
	bBEjectorsRetractPB : BOOL := FALSE;			(* Tailstock B Retract Ejectors *)

(* Screen Control *)
	bTriggerInitializeVisu: BOOL := FALSE;			(*If the Panel ID is not set then we need to go to the Initialization Screen and set it*)
	fbInitializeVisuRTRIG : R_TRIG;
	(* Screen Title Control *)
	bDisplayUnloadConf: BOOL := FALSE;				(*Display Confirm Unload*)

(* SECRET Screen*)
	bLoginPB : BOOL := FALSE;
	bLogoutPB : BOOL := FALSE;
	bASideIsLoadPB : BOOL:=FALSE;				(* Set A Side as Infeed Side Push Button *)
	bBSideIsLoadPB : BOOL:=FALSE;				(* Set B Side as Infeed Side Push Button *)

(* Test Speed Varialbes *)
	bTestSpeedOn : BOOL := FALSE;				(* Test Speed is Active *)
	nTestSpeedOverRide : UDINT := 100;			(* Current Test Speed Over-ride Value - from CX*)

END_VAR

(* Global variable list: TwinCAT_Configuration *)
(* Generated automatically by TwinCAT - (read only) *)
VAR_CONFIG
	.DriveZAWAdinputs AT %IB0 : INT;	(*  ~ {LinkedWith:TIID^Device 1 (EtherCAT)^Rack 1 Slot 0 (EK1200)^Rack 1 Slot 16 (EK1122)^Axis ZA/WA (AX5206-0000-0011)^AT 2^Digital inputs, state} *)
	.stZAAxis.PlcToNc AT %QB2277 : PLCTONC_AXIS_REF;	(*  ~ {LinkedWith:TINC^NC-Task 1 SAF^Axes^ZA Axis^Inputs^ZA Axis_FromPlc} *)
	.stZAAxis.NcToPlc AT %IB1434 : NCTOPLC_AXIS_REF;	(*  ~ {LinkedWith:TINC^NC-Task 1 SAF^Axes^ZA Axis^Outputs^ZA Axis_ToPlc} *)
	.nZAAxisDiagNumber AT %IB2 : UDINT;	(*  ~ {LinkedWith:TIID^Device 1 (EtherCAT)^Rack 1 Slot 0 (EK1200)^Rack 1 Slot 16 (EK1122)^Axis ZA/WA (AX5206-0000-0011)^AT 1^Diagnostic number} *)
	.nServoZAThrust AT %IB6 : INT;	(*  ~ {LinkedWith:TIID^Device 1 (EtherCAT)^Rack 1 Slot 0 (EK1200)^Rack 1 Slot 16 (EK1122)^Axis ZA/WA (AX5206-0000-0011)^AT 1^Torque feedback value} *)
	.stWAAxis.PlcToNc AT %QB2405 : PLCTONC_AXIS_REF;	(*  ~ {LinkedWith:TINC^NC-Task 1 SAF^Axes^WA Axis^Inputs^WA Axis_FromPlc} *)
	.stWAAxis.NcToPlc AT %IB1562 : NCTOPLC_AXIS_REF;	(*  ~ {LinkedWith:TINC^NC-Task 1 SAF^Axes^WA Axis^Outputs^WA Axis_ToPlc} *)
	.nWAAxisDiagNumber AT %IB8 : UDINT;	(*  ~ {LinkedWith:TIID^Device 1 (EtherCAT)^Rack 1 Slot 0 (EK1200)^Rack 1 Slot 16 (EK1122)^Axis ZA/WA (AX5206-0000-0011)^AT 2^Diagnostic number} *)
	.nWAAxisThrust AT %IB12 : INT;	(*  ~ {LinkedWith:TIID^Device 1 (EtherCAT)^Rack 1 Slot 0 (EK1200)^Rack 1 Slot 16 (EK1122)^Axis ZA/WA (AX5206-0000-0011)^AT 2^Torque feedback value} *)
	.nWATorqeLimitValue AT %QB0 : INT;	(*  ~ {LinkedWith:TIID^Device 1 (EtherCAT)^Rack 1 Slot 0 (EK1200)^Rack 1 Slot 16 (EK1122)^Axis ZA/WA (AX5206-0000-0011)^MDT 2^Bipolar torque limit value} *)
	.DriveZBWBdinputs AT %IB14 : INT;	(*  ~ {LinkedWith:TIID^Device 1 (EtherCAT)^Rack 1 Slot 0 (EK1200)^Rack 1 Slot 16 (EK1122)^ Axis ZB/WB (AX5206-0000-0011)^AT 2^Digital inputs, state} *)
	.stZBAxis.PlcToNc AT %QB2533 : PLCTONC_AXIS_REF;	(*  ~ {LinkedWith:TINC^NC-Task 1 SAF^Axes^ZB Axis^Inputs^ZB Axis_FromPlc} *)
	.stZBAxis.NcToPlc AT %IB1690 : NCTOPLC_AXIS_REF;	(*  ~ {LinkedWith:TINC^NC-Task 1 SAF^Axes^ZB Axis^Outputs^ZB Axis_ToPlc} *)
	.nZBAxisDiagNumber AT %IB16 : UDINT;	(*  ~ {LinkedWith:TIID^Device 1 (EtherCAT)^Rack 1 Slot 0 (EK1200)^Rack 1 Slot 16 (EK1122)^ Axis ZB/WB (AX5206-0000-0011)^AT 1^Diagnostic number} *)
	.nServoZBThrust AT %IB20 : INT;	(*  ~ {LinkedWith:TIID^Device 1 (EtherCAT)^Rack 1 Slot 0 (EK1200)^Rack 1 Slot 16 (EK1122)^ Axis ZB/WB (AX5206-0000-0011)^AT 1^Torque feedback value} *)
	.stWBAxis.PlcToNc AT %QB2661 : PLCTONC_AXIS_REF;	(*  ~ {LinkedWith:TINC^NC-Task 1 SAF^Axes^WB Axis^Inputs^WB Axis_FromPlc} *)
	.stWBAxis.NcToPlc AT %IB1818 : NCTOPLC_AXIS_REF;	(*  ~ {LinkedWith:TINC^NC-Task 1 SAF^Axes^WB Axis^Outputs^WB Axis_ToPlc} *)
	.nWBAxisDiagNumber AT %IB22 : UDINT;	(*  ~ {LinkedWith:TIID^Device 1 (EtherCAT)^Rack 1 Slot 0 (EK1200)^Rack 1 Slot 16 (EK1122)^ Axis ZB/WB (AX5206-0000-0011)^AT 2^Diagnostic number} *)
	.nWBAxisThrust AT %IB26 : INT;	(*  ~ {LinkedWith:TIID^Device 1 (EtherCAT)^Rack 1 Slot 0 (EK1200)^Rack 1 Slot 16 (EK1122)^ Axis ZB/WB (AX5206-0000-0011)^AT 2^Torque feedback value} *)
	.nWBTorqeLimitValue AT %QB2 : INT;	(*  ~ {LinkedWith:TIID^Device 1 (EtherCAT)^Rack 1 Slot 0 (EK1200)^Rack 1 Slot 16 (EK1122)^ Axis ZB/WB (AX5206-0000-0011)^MDT 2^Bipolar torque limit value} *)
	.DriveUdinputs AT %IB28 : INT;	(*  ~ {LinkedWith:TIID^Device 1 (EtherCAT)^Box 20 (CU1128)^Axis U (AX5106-0000-0011)^AT^Digital inputs, state} *)
	.stUAxis.PlcToNc AT %QB2789 : PLCTONC_AXIS_REF;	(*  ~ {LinkedWith:TINC^NC-Task 1 SAF^Axes^U Axis^Inputs^U Axis_FromPlc} *)
	.stUAxis.NcToPlc AT %IB1946 : NCTOPLC_AXIS_REF;	(*  ~ {LinkedWith:TINC^NC-Task 1 SAF^Axes^U Axis^Outputs^U Axis_ToPlc} *)
	.nUAxisDiagNumber AT %IB30 : UDINT;	(*  ~ {LinkedWith:TIID^Device 1 (EtherCAT)^Box 20 (CU1128)^Axis U (AX5106-0000-0011)^AT^Diagnostic number} *)
	.nUAxisThrust AT %IB34 : INT;	(*  ~ {LinkedWith:TIID^Device 1 (EtherCAT)^Box 20 (CU1128)^Axis U (AX5106-0000-0011)^AT^Torque feedback value} *)
	.stAxisMPG_A.PlcToNc AT %QB2917 : PLCTONC_AXIS_REF;	(*  ~ {LinkedWith:TINC^NC-Task 1 SAF^Axes^MPGA Axis^Inputs^MPGA Axis_FromPlc} *)
	.stAxisMPG_A.NcToPlc AT %IB2074 : NCTOPLC_AXIS_REF;	(*  ~ {LinkedWith:TINC^NC-Task 1 SAF^Axes^MPGA Axis^Outputs^MPGA Axis_ToPlc} *)
	.stAxisMPG_B.PlcToNc AT %QB3045 : PLCTONC_AXIS_REF;	(*  ~ {LinkedWith:TINC^NC-Task 1 SAF^Axes^MPGB Axis^Inputs^MPGB Axis_FromPlc} *)
	.stAxisMPG_B.NcToPlc AT %IB2202 : NCTOPLC_AXIS_REF;	(*  ~ {LinkedWith:TINC^NC-Task 1 SAF^Axes^MPGB Axis^Outputs^MPGB Axis_ToPlc} *)
	.fbVFD_A1.nMotorSpeed AT %IB2330 : UINT;	(*  ~ {LinkedWith:TIID^Device 1 (EtherCAT)^Box 20 (CU1128)^Rack 2 Slot 1 (EK1100)^Rack 2 Slot 8 (EK1122)^Spindle A1 (SM-EtherCAT)^Transmit PDO mapping 1^Motor Speed} *)
	.fbVFD_A1.nMotorVoltage AT %IB2332 : UINT;	(*  ~ {LinkedWith:TIID^Device 1 (EtherCAT)^Box 20 (CU1128)^Rack 2 Slot 1 (EK1100)^Rack 2 Slot 8 (EK1122)^Spindle A1 (SM-EtherCAT)^Transmit PDO mapping 1^Motor Voltage} *)
	.fbVFD_A1.nMotorCurrent AT %IB2334 : UDINT;	(*  ~ {LinkedWith:TIID^Device 1 (EtherCAT)^Box 20 (CU1128)^Rack 2 Slot 1 (EK1100)^Rack 2 Slot 8 (EK1122)^Spindle A1 (SM-EtherCAT)^Transmit PDO mapping 1^Motor Current} *)
	.fbVFD_A1.nMotorTorque AT %IB2338 : UINT;	(*  ~ {LinkedWith:TIID^Device 1 (EtherCAT)^Box 20 (CU1128)^Rack 2 Slot 1 (EK1100)^Rack 2 Slot 8 (EK1122)^Spindle A1 (SM-EtherCAT)^Transmit PDO mapping 1^Motor Torque} *)
	.fbVFD_A1.nMotorPower AT %IB2340 : UINT;	(*  ~ {LinkedWith:TIID^Device 1 (EtherCAT)^Box 20 (CU1128)^Rack 2 Slot 1 (EK1100)^Rack 2 Slot 8 (EK1122)^Spindle A1 (SM-EtherCAT)^Transmit PDO mapping 1^Motor Power} *)
	.fbVFD_A1.nDriveStatus AT %IB2342 : UINT;	(*  ~ {LinkedWith:TIID^Device 1 (EtherCAT)^Box 20 (CU1128)^Rack 2 Slot 1 (EK1100)^Rack 2 Slot 8 (EK1122)^Spindle A1 (SM-EtherCAT)^Transmit PDO mapping 2^Drive Status} *)
	.fbVFD_A1.nDCLinkVoltage AT %IB2344 : UINT;	(*  ~ {LinkedWith:TIID^Device 1 (EtherCAT)^Box 20 (CU1128)^Rack 2 Slot 1 (EK1100)^Rack 2 Slot 8 (EK1122)^Spindle A1 (SM-EtherCAT)^Transmit PDO mapping 2^DC Link Voltage} *)
	.fbVFD_A1.nOpDayCounter1 AT %IB2346 : UINT;	(*  ~ {LinkedWith:TIID^Device 1 (EtherCAT)^Box 20 (CU1128)^Rack 2 Slot 1 (EK1100)^Rack 2 Slot 8 (EK1122)^Spindle A1 (SM-EtherCAT)^Transmit PDO mapping 2^OP Day Counter #1} *)
	.fbVFD_A1.nOpDayCounter2 AT %IB2348 : UINT;	(*  ~ {LinkedWith:TIID^Device 1 (EtherCAT)^Box 20 (CU1128)^Rack 2 Slot 1 (EK1100)^Rack 2 Slot 8 (EK1122)^Spindle A1 (SM-EtherCAT)^Transmit PDO mapping 2^OP Day Counter #2} *)
	.fbVFD_A1.nEnergyCounter AT %IB2350 : INT;	(*  ~ {LinkedWith:TIID^Device 1 (EtherCAT)^Box 20 (CU1128)^Rack 2 Slot 1 (EK1100)^Rack 2 Slot 8 (EK1122)^Spindle A1 (SM-EtherCAT)^Transmit PDO mapping 2^Energy Counter kWh} *)
	.fbVFD_A1.bRunStop AT %QX3173.0 : BOOL;	(*  ~ {LinkedWith:TIID^Device 1 (EtherCAT)^Box 20 (CU1128)^Rack 2 Slot 1 (EK1100)^Rack 2 Slot 8 (EK1122)^Spindle A1 (SM-EtherCAT)^Receive PDO mapping 22^Run/Stop^Run/Stop[0]} *)
	.fbVFD_A1.bDirection AT %QX3173.1 : BOOL;	(*  ~ {LinkedWith:TIID^Device 1 (EtherCAT)^Box 20 (CU1128)^Rack 2 Slot 1 (EK1100)^Rack 2 Slot 8 (EK1122)^Spindle A1 (SM-EtherCAT)^Receive PDO mapping 22^Direction^Direction[0]} *)
	.fbVFD_A1.nSpeed AT %QB3174 : INT;	(*  ~ {LinkedWith:TIID^Device 1 (EtherCAT)^Box 20 (CU1128)^Rack 2 Slot 1 (EK1100)^Rack 2 Slot 8 (EK1122)^Spindle A1 (SM-EtherCAT)^Receive PDO mapping 22^Speed Request} *)
	.fbVFD_A1.bDriveReset AT %QX3176.0 : BOOL;	(*  ~ {LinkedWith:TIID^Device 1 (EtherCAT)^Box 20 (CU1128)^Rack 2 Slot 1 (EK1100)^Rack 2 Slot 8 (EK1122)^Spindle A1 (SM-EtherCAT)^Receive PDO mapping 22^Drive Reset^Drive Reset[0]} *)
	.bVFD_A1DataValid AT %IX1422.0 : BOOL;	(*  ~ {LinkedWith:TIID^Device 1 (EtherCAT)^Box 20 (CU1128)^Rack 2 Slot 1 (EK1100)^Rack 2 Slot 8 (EK1122)^Spindle A1 (SM-EtherCAT)^WcState^WcStateOut} *)
	.fbVFD_A2.nMotorSpeed AT %IB2352 : UINT;	(*  ~ {LinkedWith:TIID^Device 1 (EtherCAT)^Box 20 (CU1128)^Rack 2 Slot 1 (EK1100)^Rack 2 Slot 8 (EK1122)^Spindle A2 (SM-EtherCAT)^Transmit PDO mapping 1^Motor Speed} *)
	.fbVFD_A2.nMotorVoltage AT %IB2354 : UINT;	(*  ~ {LinkedWith:TIID^Device 1 (EtherCAT)^Box 20 (CU1128)^Rack 2 Slot 1 (EK1100)^Rack 2 Slot 8 (EK1122)^Spindle A2 (SM-EtherCAT)^Transmit PDO mapping 1^Motor Voltage} *)
	.fbVFD_A2.nMotorCurrent AT %IB2356 : UDINT;	(*  ~ {LinkedWith:TIID^Device 1 (EtherCAT)^Box 20 (CU1128)^Rack 2 Slot 1 (EK1100)^Rack 2 Slot 8 (EK1122)^Spindle A2 (SM-EtherCAT)^Transmit PDO mapping 1^Motor Current} *)
	.fbVFD_A2.nMotorTorque AT %IB2360 : UINT;	(*  ~ {LinkedWith:TIID^Device 1 (EtherCAT)^Box 20 (CU1128)^Rack 2 Slot 1 (EK1100)^Rack 2 Slot 8 (EK1122)^Spindle A2 (SM-EtherCAT)^Transmit PDO mapping 1^Motor Torque} *)
	.fbVFD_A2.nMotorPower AT %IB2362 : UINT;	(*  ~ {LinkedWith:TIID^Device 1 (EtherCAT)^Box 20 (CU1128)^Rack 2 Slot 1 (EK1100)^Rack 2 Slot 8 (EK1122)^Spindle A2 (SM-EtherCAT)^Transmit PDO mapping 1^Motor Power} *)
	.fbVFD_A2.nDriveStatus AT %IB2364 : UINT;	(*  ~ {LinkedWith:TIID^Device 1 (EtherCAT)^Box 20 (CU1128)^Rack 2 Slot 1 (EK1100)^Rack 2 Slot 8 (EK1122)^Spindle A2 (SM-EtherCAT)^Transmit PDO mapping 2^Drive Status} *)
	.fbVFD_A2.nDCLinkVoltage AT %IB2366 : UINT;	(*  ~ {LinkedWith:TIID^Device 1 (EtherCAT)^Box 20 (CU1128)^Rack 2 Slot 1 (EK1100)^Rack 2 Slot 8 (EK1122)^Spindle A2 (SM-EtherCAT)^Transmit PDO mapping 2^DC Link Voltage} *)
	.fbVFD_A2.nOpDayCounter1 AT %IB2368 : UINT;	(*  ~ {LinkedWith:TIID^Device 1 (EtherCAT)^Box 20 (CU1128)^Rack 2 Slot 1 (EK1100)^Rack 2 Slot 8 (EK1122)^Spindle A2 (SM-EtherCAT)^Transmit PDO mapping 2^OP Day Counter #1} *)
	.fbVFD_A2.nOpDayCounter2 AT %IB2370 : UINT;	(*  ~ {LinkedWith:TIID^Device 1 (EtherCAT)^Box 20 (CU1128)^Rack 2 Slot 1 (EK1100)^Rack 2 Slot 8 (EK1122)^Spindle A2 (SM-EtherCAT)^Transmit PDO mapping 2^OP Day Counter #2} *)
	.fbVFD_A2.nEnergyCounter AT %IB2372 : INT;	(*  ~ {LinkedWith:TIID^Device 1 (EtherCAT)^Box 20 (CU1128)^Rack 2 Slot 1 (EK1100)^Rack 2 Slot 8 (EK1122)^Spindle A2 (SM-EtherCAT)^Transmit PDO mapping 2^Energy Counter kWh} *)
	.fbVFD_A2.bRunStop AT %QX3176.1 : BOOL;	(*  ~ {LinkedWith:TIID^Device 1 (EtherCAT)^Box 20 (CU1128)^Rack 2 Slot 1 (EK1100)^Rack 2 Slot 8 (EK1122)^Spindle A2 (SM-EtherCAT)^Receive PDO mapping 22^Run/Stop^Run/Stop[0]} *)
	.fbVFD_A2.bDirection AT %QX3176.2 : BOOL;	(*  ~ {LinkedWith:TIID^Device 1 (EtherCAT)^Box 20 (CU1128)^Rack 2 Slot 1 (EK1100)^Rack 2 Slot 8 (EK1122)^Spindle A2 (SM-EtherCAT)^Receive PDO mapping 22^Direction^Direction[0]} *)
	.fbVFD_A2.nSpeed AT %QB3177 : INT;	(*  ~ {LinkedWith:TIID^Device 1 (EtherCAT)^Box 20 (CU1128)^Rack 2 Slot 1 (EK1100)^Rack 2 Slot 8 (EK1122)^Spindle A2 (SM-EtherCAT)^Receive PDO mapping 22^Speed Request} *)
	.fbVFD_A2.bDriveReset AT %QX3179.0 : BOOL;	(*  ~ {LinkedWith:TIID^Device 1 (EtherCAT)^Box 20 (CU1128)^Rack 2 Slot 1 (EK1100)^Rack 2 Slot 8 (EK1122)^Spindle A2 (SM-EtherCAT)^Receive PDO mapping 22^Drive Reset^Drive Reset[0]} *)
	.bVFD_A2DataValid AT %IX1422.1 : BOOL;	(*  ~ {LinkedWith:TIID^Device 1 (EtherCAT)^Box 20 (CU1128)^Rack 2 Slot 1 (EK1100)^Rack 2 Slot 8 (EK1122)^Spindle A2 (SM-EtherCAT)^WcState^WcStateOut} *)
	.fbVFD_A3.nMotorSpeed AT %IB2374 : UINT;	(*  ~ {LinkedWith:TIID^Device 1 (EtherCAT)^Box 20 (CU1128)^Rack 2 Slot 1 (EK1100)^Rack 2 Slot 8 (EK1122)^Spindle A3 (SM-EtherCAT)^Transmit PDO mapping 1^Motor Speed} *)
	.fbVFD_A3.nMotorVoltage AT %IB2376 : UINT;	(*  ~ {LinkedWith:TIID^Device 1 (EtherCAT)^Box 20 (CU1128)^Rack 2 Slot 1 (EK1100)^Rack 2 Slot 8 (EK1122)^Spindle A3 (SM-EtherCAT)^Transmit PDO mapping 1^Motor Voltage} *)
	.fbVFD_A3.nMotorCurrent AT %IB2378 : UDINT;	(*  ~ {LinkedWith:TIID^Device 1 (EtherCAT)^Box 20 (CU1128)^Rack 2 Slot 1 (EK1100)^Rack 2 Slot 8 (EK1122)^Spindle A3 (SM-EtherCAT)^Transmit PDO mapping 1^Motor Current} *)
	.fbVFD_A3.nMotorTorque AT %IB2382 : UINT;	(*  ~ {LinkedWith:TIID^Device 1 (EtherCAT)^Box 20 (CU1128)^Rack 2 Slot 1 (EK1100)^Rack 2 Slot 8 (EK1122)^Spindle A3 (SM-EtherCAT)^Transmit PDO mapping 1^Motor Torque} *)
	.fbVFD_A3.nMotorPower AT %IB2384 : UINT;	(*  ~ {LinkedWith:TIID^Device 1 (EtherCAT)^Box 20 (CU1128)^Rack 2 Slot 1 (EK1100)^Rack 2 Slot 8 (EK1122)^Spindle A3 (SM-EtherCAT)^Transmit PDO mapping 1^Motor Power} *)
	.fbVFD_A3.nDriveStatus AT %IB2386 : UINT;	(*  ~ {LinkedWith:TIID^Device 1 (EtherCAT)^Box 20 (CU1128)^Rack 2 Slot 1 (EK1100)^Rack 2 Slot 8 (EK1122)^Spindle A3 (SM-EtherCAT)^Transmit PDO mapping 2^Drive Status} *)
	.fbVFD_A3.nDCLinkVoltage AT %IB2388 : UINT;	(*  ~ {LinkedWith:TIID^Device 1 (EtherCAT)^Box 20 (CU1128)^Rack 2 Slot 1 (EK1100)^Rack 2 Slot 8 (EK1122)^Spindle A3 (SM-EtherCAT)^Transmit PDO mapping 2^DC Link Voltage} *)
	.fbVFD_A3.nOpDayCounter1 AT %IB2390 : UINT;	(*  ~ {LinkedWith:TIID^Device 1 (EtherCAT)^Box 20 (CU1128)^Rack 2 Slot 1 (EK1100)^Rack 2 Slot 8 (EK1122)^Spindle A3 (SM-EtherCAT)^Transmit PDO mapping 2^OP Day Counter #1} *)
	.fbVFD_A3.nOpDayCounter2 AT %IB2392 : UINT;	(*  ~ {LinkedWith:TIID^Device 1 (EtherCAT)^Box 20 (CU1128)^Rack 2 Slot 1 (EK1100)^Rack 2 Slot 8 (EK1122)^Spindle A3 (SM-EtherCAT)^Transmit PDO mapping 2^OP Day Counter #2} *)
	.fbVFD_A3.nEnergyCounter AT %IB2394 : INT;	(*  ~ {LinkedWith:TIID^Device 1 (EtherCAT)^Box 20 (CU1128)^Rack 2 Slot 1 (EK1100)^Rack 2 Slot 8 (EK1122)^Spindle A3 (SM-EtherCAT)^Transmit PDO mapping 2^Energy Counter kWh} *)
	.fbVFD_A3.bRunStop AT %QX3179.1 : BOOL;	(*  ~ {LinkedWith:TIID^Device 1 (EtherCAT)^Box 20 (CU1128)^Rack 2 Slot 1 (EK1100)^Rack 2 Slot 8 (EK1122)^Spindle A3 (SM-EtherCAT)^Receive PDO mapping 22^Run/Stop^Run/Stop[0]} *)
	.fbVFD_A3.bDirection AT %QX3179.2 : BOOL;	(*  ~ {LinkedWith:TIID^Device 1 (EtherCAT)^Box 20 (CU1128)^Rack 2 Slot 1 (EK1100)^Rack 2 Slot 8 (EK1122)^Spindle A3 (SM-EtherCAT)^Receive PDO mapping 22^Direction^Direction[0]} *)
	.fbVFD_A3.nSpeed AT %QB3180 : INT;	(*  ~ {LinkedWith:TIID^Device 1 (EtherCAT)^Box 20 (CU1128)^Rack 2 Slot 1 (EK1100)^Rack 2 Slot 8 (EK1122)^Spindle A3 (SM-EtherCAT)^Receive PDO mapping 22^Speed Request} *)
	.fbVFD_A3.bDriveReset AT %QX3182.0 : BOOL;	(*  ~ {LinkedWith:TIID^Device 1 (EtherCAT)^Box 20 (CU1128)^Rack 2 Slot 1 (EK1100)^Rack 2 Slot 8 (EK1122)^Spindle A3 (SM-EtherCAT)^Receive PDO mapping 22^Drive Reset^Drive Reset[0]} *)
	.bVFD_A3DataValid AT %IX1422.2 : BOOL;	(*  ~ {LinkedWith:TIID^Device 1 (EtherCAT)^Box 20 (CU1128)^Rack 2 Slot 1 (EK1100)^Rack 2 Slot 8 (EK1122)^Spindle A3 (SM-EtherCAT)^WcState^WcStateOut} *)
	.fbVFD_B1.nMotorSpeed AT %IB2396 : UINT;	(*  ~ {LinkedWith:TIID^Device 1 (EtherCAT)^Box 20 (CU1128)^Rack 2 Slot 1 (EK1100)^Rack 2 Slot 8 (EK1122)^Spindle B1 (SM-EtherCAT)^Transmit PDO mapping 1^Motor Speed} *)
	.fbVFD_B1.nMotorVoltage AT %IB2398 : UINT;	(*  ~ {LinkedWith:TIID^Device 1 (EtherCAT)^Box 20 (CU1128)^Rack 2 Slot 1 (EK1100)^Rack 2 Slot 8 (EK1122)^Spindle B1 (SM-EtherCAT)^Transmit PDO mapping 1^Motor Voltage} *)
	.fbVFD_B1.nMotorCurrent AT %IB2400 : UDINT;	(*  ~ {LinkedWith:TIID^Device 1 (EtherCAT)^Box 20 (CU1128)^Rack 2 Slot 1 (EK1100)^Rack 2 Slot 8 (EK1122)^Spindle B1 (SM-EtherCAT)^Transmit PDO mapping 1^Motor Current} *)
	.fbVFD_B1.nMotorTorque AT %IB2404 : UINT;	(*  ~ {LinkedWith:TIID^Device 1 (EtherCAT)^Box 20 (CU1128)^Rack 2 Slot 1 (EK1100)^Rack 2 Slot 8 (EK1122)^Spindle B1 (SM-EtherCAT)^Transmit PDO mapping 1^Motor Torque} *)
	.fbVFD_B1.nMotorPower AT %IB2406 : UINT;	(*  ~ {LinkedWith:TIID^Device 1 (EtherCAT)^Box 20 (CU1128)^Rack 2 Slot 1 (EK1100)^Rack 2 Slot 8 (EK1122)^Spindle B1 (SM-EtherCAT)^Transmit PDO mapping 1^Motor Power} *)
	.fbVFD_B1.nDriveStatus AT %IB2408 : UINT;	(*  ~ {LinkedWith:TIID^Device 1 (EtherCAT)^Box 20 (CU1128)^Rack 2 Slot 1 (EK1100)^Rack 2 Slot 8 (EK1122)^Spindle B1 (SM-EtherCAT)^Transmit PDO mapping 2^Drive Status} *)
	.fbVFD_B1.nDCLinkVoltage AT %IB2410 : UINT;	(*  ~ {LinkedWith:TIID^Device 1 (EtherCAT)^Box 20 (CU1128)^Rack 2 Slot 1 (EK1100)^Rack 2 Slot 8 (EK1122)^Spindle B1 (SM-EtherCAT)^Transmit PDO mapping 2^DC Link Voltage} *)
	.fbVFD_B1.nOpDayCounter1 AT %IB2412 : UINT;	(*  ~ {LinkedWith:TIID^Device 1 (EtherCAT)^Box 20 (CU1128)^Rack 2 Slot 1 (EK1100)^Rack 2 Slot 8 (EK1122)^Spindle B1 (SM-EtherCAT)^Transmit PDO mapping 2^OP Day Counter #1} *)
	.fbVFD_B1.nOpDayCounter2 AT %IB2414 : UINT;	(*  ~ {LinkedWith:TIID^Device 1 (EtherCAT)^Box 20 (CU1128)^Rack 2 Slot 1 (EK1100)^Rack 2 Slot 8 (EK1122)^Spindle B1 (SM-EtherCAT)^Transmit PDO mapping 2^OP Day Counter #2} *)
	.fbVFD_B1.nEnergyCounter AT %IB2416 : INT;	(*  ~ {LinkedWith:TIID^Device 1 (EtherCAT)^Box 20 (CU1128)^Rack 2 Slot 1 (EK1100)^Rack 2 Slot 8 (EK1122)^Spindle B1 (SM-EtherCAT)^Transmit PDO mapping 2^Energy Counter kWh} *)
	.fbVFD_B1.bRunStop AT %QX3182.1 : BOOL;	(*  ~ {LinkedWith:TIID^Device 1 (EtherCAT)^Box 20 (CU1128)^Rack 2 Slot 1 (EK1100)^Rack 2 Slot 8 (EK1122)^Spindle B1 (SM-EtherCAT)^Receive PDO mapping 22^Run/Stop^Run/Stop[0]} *)
	.fbVFD_B1.bDirection AT %QX3182.2 : BOOL;	(*  ~ {LinkedWith:TIID^Device 1 (EtherCAT)^Box 20 (CU1128)^Rack 2 Slot 1 (EK1100)^Rack 2 Slot 8 (EK1122)^Spindle B1 (SM-EtherCAT)^Receive PDO mapping 22^Direction^Direction[0]} *)
	.fbVFD_B1.nSpeed AT %QB3183 : INT;	(*  ~ {LinkedWith:TIID^Device 1 (EtherCAT)^Box 20 (CU1128)^Rack 2 Slot 1 (EK1100)^Rack 2 Slot 8 (EK1122)^Spindle B1 (SM-EtherCAT)^Receive PDO mapping 22^Speed Request} *)
	.fbVFD_B1.bDriveReset AT %QX3185.0 : BOOL;	(*  ~ {LinkedWith:TIID^Device 1 (EtherCAT)^Box 20 (CU1128)^Rack 2 Slot 1 (EK1100)^Rack 2 Slot 8 (EK1122)^Spindle B1 (SM-EtherCAT)^Receive PDO mapping 22^Drive Reset^Drive Reset[0]} *)
	.bVFD_B1DataValid AT %IX1422.3 : BOOL;	(*  ~ {LinkedWith:TIID^Device 1 (EtherCAT)^Box 20 (CU1128)^Rack 2 Slot 1 (EK1100)^Rack 2 Slot 8 (EK1122)^Spindle B1 (SM-EtherCAT)^WcState^WcStateOut} *)
	.fbVFD_B2.nMotorSpeed AT %IB2418 : UINT;	(*  ~ {LinkedWith:TIID^Device 1 (EtherCAT)^Box 20 (CU1128)^Rack 2 Slot 1 (EK1100)^Rack 2 Slot 8 (EK1122)^Spindle B2 (SM-EtherCAT)^Transmit PDO mapping 1^Motor Speed} *)
	.fbVFD_B2.nMotorVoltage AT %IB2420 : UINT;	(*  ~ {LinkedWith:TIID^Device 1 (EtherCAT)^Box 20 (CU1128)^Rack 2 Slot 1 (EK1100)^Rack 2 Slot 8 (EK1122)^Spindle B2 (SM-EtherCAT)^Transmit PDO mapping 1^Motor Voltage} *)
	.fbVFD_B2.nMotorCurrent AT %IB2422 : UDINT;	(*  ~ {LinkedWith:TIID^Device 1 (EtherCAT)^Box 20 (CU1128)^Rack 2 Slot 1 (EK1100)^Rack 2 Slot 8 (EK1122)^Spindle B2 (SM-EtherCAT)^Transmit PDO mapping 1^Motor Current} *)
	.fbVFD_B2.nMotorTorque AT %IB2426 : UINT;	(*  ~ {LinkedWith:TIID^Device 1 (EtherCAT)^Box 20 (CU1128)^Rack 2 Slot 1 (EK1100)^Rack 2 Slot 8 (EK1122)^Spindle B2 (SM-EtherCAT)^Transmit PDO mapping 1^Motor Torque} *)
	.fbVFD_B2.nMotorPower AT %IB2428 : UINT;	(*  ~ {LinkedWith:TIID^Device 1 (EtherCAT)^Box 20 (CU1128)^Rack 2 Slot 1 (EK1100)^Rack 2 Slot 8 (EK1122)^Spindle B2 (SM-EtherCAT)^Transmit PDO mapping 1^Motor Power} *)
	.fbVFD_B2.nDriveStatus AT %IB2430 : UINT;	(*  ~ {LinkedWith:TIID^Device 1 (EtherCAT)^Box 20 (CU1128)^Rack 2 Slot 1 (EK1100)^Rack 2 Slot 8 (EK1122)^Spindle B2 (SM-EtherCAT)^Transmit PDO mapping 2^Drive Status} *)
	.fbVFD_B2.nDCLinkVoltage AT %IB2432 : UINT;	(*  ~ {LinkedWith:TIID^Device 1 (EtherCAT)^Box 20 (CU1128)^Rack 2 Slot 1 (EK1100)^Rack 2 Slot 8 (EK1122)^Spindle B2 (SM-EtherCAT)^Transmit PDO mapping 2^DC Link Voltage} *)
	.fbVFD_B2.nOpDayCounter1 AT %IB2434 : UINT;	(*  ~ {LinkedWith:TIID^Device 1 (EtherCAT)^Box 20 (CU1128)^Rack 2 Slot 1 (EK1100)^Rack 2 Slot 8 (EK1122)^Spindle B2 (SM-EtherCAT)^Transmit PDO mapping 2^OP Day Counter #1} *)
	.fbVFD_B2.nOpDayCounter2 AT %IB2436 : UINT;	(*  ~ {LinkedWith:TIID^Device 1 (EtherCAT)^Box 20 (CU1128)^Rack 2 Slot 1 (EK1100)^Rack 2 Slot 8 (EK1122)^Spindle B2 (SM-EtherCAT)^Transmit PDO mapping 2^OP Day Counter #2} *)
	.fbVFD_B2.nEnergyCounter AT %IB2438 : INT;	(*  ~ {LinkedWith:TIID^Device 1 (EtherCAT)^Box 20 (CU1128)^Rack 2 Slot 1 (EK1100)^Rack 2 Slot 8 (EK1122)^Spindle B2 (SM-EtherCAT)^Transmit PDO mapping 2^Energy Counter kWh} *)
	.fbVFD_B2.bRunStop AT %QX3185.1 : BOOL;	(*  ~ {LinkedWith:TIID^Device 1 (EtherCAT)^Box 20 (CU1128)^Rack 2 Slot 1 (EK1100)^Rack 2 Slot 8 (EK1122)^Spindle B2 (SM-EtherCAT)^Receive PDO mapping 22^Run/Stop^Run/Stop[0]} *)
	.fbVFD_B2.bDirection AT %QX3185.2 : BOOL;	(*  ~ {LinkedWith:TIID^Device 1 (EtherCAT)^Box 20 (CU1128)^Rack 2 Slot 1 (EK1100)^Rack 2 Slot 8 (EK1122)^Spindle B2 (SM-EtherCAT)^Receive PDO mapping 22^Direction^Direction[0]} *)
	.fbVFD_B2.nSpeed AT %QB3186 : INT;	(*  ~ {LinkedWith:TIID^Device 1 (EtherCAT)^Box 20 (CU1128)^Rack 2 Slot 1 (EK1100)^Rack 2 Slot 8 (EK1122)^Spindle B2 (SM-EtherCAT)^Receive PDO mapping 22^Speed Request} *)
	.fbVFD_B2.bDriveReset AT %QX3188.0 : BOOL;	(*  ~ {LinkedWith:TIID^Device 1 (EtherCAT)^Box 20 (CU1128)^Rack 2 Slot 1 (EK1100)^Rack 2 Slot 8 (EK1122)^Spindle B2 (SM-EtherCAT)^Receive PDO mapping 22^Drive Reset^Drive Reset[0]} *)
	.bVFD_B2DataValid AT %IX1422.4 : BOOL;	(*  ~ {LinkedWith:TIID^Device 1 (EtherCAT)^Box 20 (CU1128)^Rack 2 Slot 1 (EK1100)^Rack 2 Slot 8 (EK1122)^Spindle B2 (SM-EtherCAT)^WcState^WcStateOut} *)
	.fbVFD_B3.nMotorSpeed AT %IB2440 : UINT;	(*  ~ {LinkedWith:TIID^Device 1 (EtherCAT)^Box 20 (CU1128)^Rack 2 Slot 1 (EK1100)^Rack 2 Slot 8 (EK1122)^Spindle B3 (SM-EtherCAT)^Transmit PDO mapping 1^Motor Speed} *)
	.fbVFD_B3.nMotorVoltage AT %IB2442 : UINT;	(*  ~ {LinkedWith:TIID^Device 1 (EtherCAT)^Box 20 (CU1128)^Rack 2 Slot 1 (EK1100)^Rack 2 Slot 8 (EK1122)^Spindle B3 (SM-EtherCAT)^Transmit PDO mapping 1^Motor Voltage} *)
	.fbVFD_B3.nMotorCurrent AT %IB2444 : UDINT;	(*  ~ {LinkedWith:TIID^Device 1 (EtherCAT)^Box 20 (CU1128)^Rack 2 Slot 1 (EK1100)^Rack 2 Slot 8 (EK1122)^Spindle B3 (SM-EtherCAT)^Transmit PDO mapping 1^Motor Current} *)
	.fbVFD_B3.nMotorTorque AT %IB2448 : UINT;	(*  ~ {LinkedWith:TIID^Device 1 (EtherCAT)^Box 20 (CU1128)^Rack 2 Slot 1 (EK1100)^Rack 2 Slot 8 (EK1122)^Spindle B3 (SM-EtherCAT)^Transmit PDO mapping 1^Motor Torque} *)
	.fbVFD_B3.nMotorPower AT %IB2450 : UINT;	(*  ~ {LinkedWith:TIID^Device 1 (EtherCAT)^Box 20 (CU1128)^Rack 2 Slot 1 (EK1100)^Rack 2 Slot 8 (EK1122)^Spindle B3 (SM-EtherCAT)^Transmit PDO mapping 1^Motor Power} *)
	.fbVFD_B3.nDriveStatus AT %IB2452 : UINT;	(*  ~ {LinkedWith:TIID^Device 1 (EtherCAT)^Box 20 (CU1128)^Rack 2 Slot 1 (EK1100)^Rack 2 Slot 8 (EK1122)^Spindle B3 (SM-EtherCAT)^Transmit PDO mapping 2^Drive Status} *)
	.fbVFD_B3.nDCLinkVoltage AT %IB2454 : UINT;	(*  ~ {LinkedWith:TIID^Device 1 (EtherCAT)^Box 20 (CU1128)^Rack 2 Slot 1 (EK1100)^Rack 2 Slot 8 (EK1122)^Spindle B3 (SM-EtherCAT)^Transmit PDO mapping 2^DC Link Voltage} *)
	.fbVFD_B3.nOpDayCounter1 AT %IB2456 : UINT;	(*  ~ {LinkedWith:TIID^Device 1 (EtherCAT)^Box 20 (CU1128)^Rack 2 Slot 1 (EK1100)^Rack 2 Slot 8 (EK1122)^Spindle B3 (SM-EtherCAT)^Transmit PDO mapping 2^OP Day Counter #1} *)
	.fbVFD_B3.nOpDayCounter2 AT %IB2458 : UINT;	(*  ~ {LinkedWith:TIID^Device 1 (EtherCAT)^Box 20 (CU1128)^Rack 2 Slot 1 (EK1100)^Rack 2 Slot 8 (EK1122)^Spindle B3 (SM-EtherCAT)^Transmit PDO mapping 2^OP Day Counter #2} *)
	.fbVFD_B3.nEnergyCounter AT %IB2460 : INT;	(*  ~ {LinkedWith:TIID^Device 1 (EtherCAT)^Box 20 (CU1128)^Rack 2 Slot 1 (EK1100)^Rack 2 Slot 8 (EK1122)^Spindle B3 (SM-EtherCAT)^Transmit PDO mapping 2^Energy Counter kWh} *)
	.fbVFD_B3.bRunStop AT %QX3188.1 : BOOL;	(*  ~ {LinkedWith:TIID^Device 1 (EtherCAT)^Box 20 (CU1128)^Rack 2 Slot 1 (EK1100)^Rack 2 Slot 8 (EK1122)^Spindle B3 (SM-EtherCAT)^Receive PDO mapping 22^Run/Stop^Run/Stop[0]} *)
	.fbVFD_B3.bDirection AT %QX3188.2 : BOOL;	(*  ~ {LinkedWith:TIID^Device 1 (EtherCAT)^Box 20 (CU1128)^Rack 2 Slot 1 (EK1100)^Rack 2 Slot 8 (EK1122)^Spindle B3 (SM-EtherCAT)^Receive PDO mapping 22^Direction^Direction[0]} *)
	.fbVFD_B3.nSpeed AT %QB3189 : INT;	(*  ~ {LinkedWith:TIID^Device 1 (EtherCAT)^Box 20 (CU1128)^Rack 2 Slot 1 (EK1100)^Rack 2 Slot 8 (EK1122)^Spindle B3 (SM-EtherCAT)^Receive PDO mapping 22^Speed Request} *)
	.fbVFD_B3.bDriveReset AT %QX3191.0 : BOOL;	(*  ~ {LinkedWith:TIID^Device 1 (EtherCAT)^Box 20 (CU1128)^Rack 2 Slot 1 (EK1100)^Rack 2 Slot 8 (EK1122)^Spindle B3 (SM-EtherCAT)^Receive PDO mapping 22^Drive Reset^Drive Reset[0]} *)
	.bVFD_B3DataValid AT %IX1422.5 : BOOL;	(*  ~ {LinkedWith:TIID^Device 1 (EtherCAT)^Box 20 (CU1128)^Rack 2 Slot 1 (EK1100)^Rack 2 Slot 8 (EK1122)^Spindle B3 (SM-EtherCAT)^WcState^WcStateOut} *)
	.nVFD_A1Addr AT %IB36 : UINT;	(*  ~ {LinkedWith:TIID^Device 1 (EtherCAT)^Box 20 (CU1128)^Rack 2 Slot 1 (EK1100)^Rack 2 Slot 8 (EK1122)^Spindle A1 (SM-EtherCAT)^InfoData^AdsAddr^port} *)
	.nVFD_A2Addr AT %IB38 : UINT;	(*  ~ {LinkedWith:TIID^Device 1 (EtherCAT)^Box 20 (CU1128)^Rack 2 Slot 1 (EK1100)^Rack 2 Slot 8 (EK1122)^Spindle A2 (SM-EtherCAT)^InfoData^AdsAddr^port} *)
	.nVFD_A3Addr AT %IB40 : UINT;	(*  ~ {LinkedWith:TIID^Device 1 (EtherCAT)^Box 20 (CU1128)^Rack 2 Slot 1 (EK1100)^Rack 2 Slot 8 (EK1122)^Spindle A3 (SM-EtherCAT)^InfoData^AdsAddr^port} *)
	.nVFD_B1Addr AT %IB42 : UINT;	(*  ~ {LinkedWith:TIID^Device 1 (EtherCAT)^Box 20 (CU1128)^Rack 2 Slot 1 (EK1100)^Rack 2 Slot 8 (EK1122)^Spindle B1 (SM-EtherCAT)^InfoData^AdsAddr^port} *)
	.nVFD_B2Addr AT %IB44 : UINT;	(*  ~ {LinkedWith:TIID^Device 1 (EtherCAT)^Box 20 (CU1128)^Rack 2 Slot 1 (EK1100)^Rack 2 Slot 8 (EK1122)^Spindle B2 (SM-EtherCAT)^InfoData^AdsAddr^port} *)
	.nVFD_B3Addr AT %IB46 : UINT;	(*  ~ {LinkedWith:TIID^Device 1 (EtherCAT)^Box 20 (CU1128)^Rack 2 Slot 1 (EK1100)^Rack 2 Slot 8 (EK1122)^Spindle B3 (SM-EtherCAT)^InfoData^AdsAddr^port} *)
	.bPB1AConfirm AT %IX1422.6 : BOOL;	(*  ~ {LinkedWith:TIID^Device 1 (EtherCAT)^Rack 1 Slot 0 (EK1200)^Rack 1 Slot 1 (EL1809)^Channel 1^Input} *)
	.bPB2ACycleStart AT %IX1422.7 : BOOL;	(*  ~ {LinkedWith:TIID^Device 1 (EtherCAT)^Rack 1 Slot 0 (EK1200)^Rack 1 Slot 1 (EL1809)^Channel 2^Input} *)
	.bPB3ACycleCommon AT %IX1423.0 : BOOL;	(*  ~ {LinkedWith:TIID^Device 1 (EtherCAT)^Rack 1 Slot 0 (EK1200)^Rack 1 Slot 1 (EL1809)^Channel 3^Input} *)
	.bPB4ADrillReturn AT %IX1423.1 : BOOL;	(*  ~ {LinkedWith:TIID^Device 1 (EtherCAT)^Rack 1 Slot 0 (EK1200)^Rack 1 Slot 1 (EL1809)^Channel 4^Input} *)
	.bPB1BConfirm AT %IX1423.2 : BOOL;	(*  ~ {LinkedWith:TIID^Device 1 (EtherCAT)^Rack 1 Slot 0 (EK1200)^Rack 1 Slot 1 (EL1809)^Channel 5^Input} *)
	.bPB2BCycleStart AT %IX1423.3 : BOOL;	(*  ~ {LinkedWith:TIID^Device 1 (EtherCAT)^Rack 1 Slot 0 (EK1200)^Rack 1 Slot 1 (EL1809)^Channel 6^Input} *)
	.bPB3BCycleCommon AT %IX1423.4 : BOOL;	(*  ~ {LinkedWith:TIID^Device 1 (EtherCAT)^Rack 1 Slot 0 (EK1200)^Rack 1 Slot 1 (EL1809)^Channel 7^Input} *)
	.bPB4BDrillReturn AT %IX1423.5 : BOOL;	(*  ~ {LinkedWith:TIID^Device 1 (EtherCAT)^Rack 1 Slot 0 (EK1200)^Rack 1 Slot 1 (EL1809)^Channel 8^Input} *)
	.bChipConveyorVFDFault AT %IX1423.6 : BOOL;
	.bCleanTankLevel AT %IX1423.7 : BOOL;	(*  ~ {LinkedWith:TIID^Device 1 (EtherCAT)^Rack 1 Slot 0 (EK1200)^Rack 1 Slot 1 (EL1809)^Channel 11^Input} *)
	.bCoolantTankOverflow AT %IX1424.0 : BOOL;	(*  ~ {LinkedWith:TIID^Device 1 (EtherCAT)^Rack 1 Slot 0 (EK1200)^Rack 1 Slot 1 (EL1809)^Channel 12^Input} *)
	.bFilter1Dirty AT %IX1424.1 : BOOL;	(*  ~ {LinkedWith:TIID^Device 1 (EtherCAT)^Rack 1 Slot 0 (EK1200)^Rack 1 Slot 1 (EL1809)^Channel 13^Input} *)
	.bFilter2Dirty AT %IX1424.2 : BOOL;	(*  ~ {LinkedWith:TIID^Device 1 (EtherCAT)^Rack 1 Slot 0 (EK1200)^Rack 1 Slot 1 (EL1809)^Channel 14^Input} *)
	.bFilter3Dirty AT %IX1424.3 : BOOL;	(*  ~ {LinkedWith:TIID^Device 1 (EtherCAT)^Rack 1 Slot 0 (EK1200)^Rack 1 Slot 1 (EL1809)^Channel 15^Input} *)
	.bFilter4Dirty AT %IX1424.4 : BOOL;	(*  ~ {LinkedWith:TIID^Device 1 (EtherCAT)^Rack 1 Slot 0 (EK1200)^Rack 1 Slot 1 (EL1809)^Channel 16^Input} *)
	.bACoolantPressure AT %IX1424.5 : BOOL;	(*  ~ {LinkedWith:TIID^Device 1 (EtherCAT)^Rack 1 Slot 0 (EK1200)^Rack 1 Slot 2 (EL1809)^Channel 1^Input} *)
	.bBCoolantPressure AT %IX1424.6 : BOOL;	(*  ~ {LinkedWith:TIID^Device 1 (EtherCAT)^Rack 1 Slot 0 (EK1200)^Rack 1 Slot 2 (EL1809)^Channel 2^Input} *)
	.bLubeLevel AT %IX1424.7 : BOOL;	(*  ~ {LinkedWith:TIID^Device 1 (EtherCAT)^Rack 1 Slot 0 (EK1200)^Rack 1 Slot 2 (EL1809)^Channel 3^Input} *)
	.bLubePressure AT %IX1425.0 : BOOL;	(*  ~ {LinkedWith:TIID^Device 1 (EtherCAT)^Rack 1 Slot 0 (EK1200)^Rack 1 Slot 2 (EL1809)^Channel 4^Input} *)
	.bHydraulicSystemLevel AT %IX1425.1 : BOOL;	(*  ~ {LinkedWith:TIID^Device 1 (EtherCAT)^Rack 1 Slot 0 (EK1200)^Rack 1 Slot 2 (EL1809)^Channel 5^Input} *)
	.bHydraulicSystemPressure AT %IX1425.2 : BOOL;	(*  ~ {LinkedWith:TIID^Device 1 (EtherCAT)^Rack 1 Slot 0 (EK1200)^Rack 1 Slot 2 (EL1809)^Channel 6^Input} *)
	.bHydraulicTemperature AT %IX1425.3 : BOOL;	(*  ~ {LinkedWith:TIID^Device 1 (EtherCAT)^Rack 1 Slot 0 (EK1200)^Rack 1 Slot 2 (EL1809)^Channel 7^Input} *)
	.bPneumaticSystemPressure AT %IX1425.4 : BOOL;	(*  ~ {LinkedWith:TIID^Device 1 (EtherCAT)^Rack 1 Slot 0 (EK1200)^Rack 1 Slot 2 (EL1809)^Channel 9^Input} *)
	.bMCC_SConfirm AT %IX1425.5 : BOOL;	(*  ~ {LinkedWith:TIID^Device 1 (EtherCAT)^Rack 1 Slot 0 (EK1200)^Rack 1 Slot 2 (EL1809)^Channel 11^Input} *)
	.bMCR AT %IX1425.6 : BOOL;	(*  ~ {LinkedWith:TIID^Device 1 (EtherCAT)^Rack 1 Slot 0 (EK1200)^Rack 1 Slot 2 (EL1809)^Channel 16^Input} *)
	.nCoolantTemp AT %IB48 : INT;	(*  ~ {LinkedWith:TIID^Device 1 (EtherCAT)^Rack 1 Slot 0 (EK1200)^Rack 1 Slot 4 (EL3311)^TC Inputs^Value} *)
	.nSpindleTachA1 AT %IB50 : INT;	(*  ~ {LinkedWith:TIID^Device 1 (EtherCAT)^Rack 1 Slot 0 (EK1200)^Rack 1 Slot 7 (EL3152)^Channel 1^Value} *)
	.nCoolantFlowA1 AT %IB52 : INT;	(*  ~ {LinkedWith:TIID^Device 1 (EtherCAT)^Rack 1 Slot 0 (EK1200)^Rack 1 Slot 7 (EL3152)^Channel 2^Value} *)
	.nSpindleTachA2 AT %IB54 : INT;	(*  ~ {LinkedWith:TIID^Device 1 (EtherCAT)^Rack 1 Slot 0 (EK1200)^Rack 1 Slot 8(EL3152)^Channel 1^Value} *)
	.nCoolantFlowA2 AT %IB56 : INT;	(*  ~ {LinkedWith:TIID^Device 1 (EtherCAT)^Rack 1 Slot 0 (EK1200)^Rack 1 Slot 8(EL3152)^Channel 2^Value} *)
	.nSpindleTachA3 AT %IB58 : INT;	(*  ~ {LinkedWith:TIID^Device 1 (EtherCAT)^Rack 1 Slot 0 (EK1200)^Rack 1 Slot 9 (EL3152)^Channel 1^Value} *)
	.nCoolantFlowA3 AT %IB60 : INT;	(*  ~ {LinkedWith:TIID^Device 1 (EtherCAT)^Rack 1 Slot 0 (EK1200)^Rack 1 Slot 9 (EL3152)^Channel 2^Value} *)
	.nSpindleTachB1 AT %IB62 : INT;	(*  ~ {LinkedWith:TIID^Device 1 (EtherCAT)^Rack 1 Slot 0 (EK1200)^Rack 1 Slot 11 (EL3152)^Channel 1^Value} *)
	.nCoolantFlowB1 AT %IB64 : INT;	(*  ~ {LinkedWith:TIID^Device 1 (EtherCAT)^Rack 1 Slot 0 (EK1200)^Rack 1 Slot 11 (EL3152)^Channel 2^Value} *)
	.nSpindleTachB2 AT %IB66 : INT;	(*  ~ {LinkedWith:TIID^Device 1 (EtherCAT)^Rack 1 Slot 0 (EK1200)^Rack 1 Slot 12 (EL3152)^Channel 1^Value} *)
	.nCoolantFlowB2 AT %IB68 : INT;	(*  ~ {LinkedWith:TIID^Device 1 (EtherCAT)^Rack 1 Slot 0 (EK1200)^Rack 1 Slot 12 (EL3152)^Channel 2^Value} *)
	.nSpindleTachB3 AT %IB70 : INT;	(*  ~ {LinkedWith:TIID^Device 1 (EtherCAT)^Rack 1 Slot 0 (EK1200)^Rack 1 Slot 13 (EL3152)^Channel 1^Value} *)
	.nCoolantFlowB3 AT %IB72 : INT;	(*  ~ {LinkedWith:TIID^Device 1 (EtherCAT)^Rack 1 Slot 0 (EK1200)^Rack 1 Slot 13 (EL3152)^Channel 2^Value} *)
	.bZAAxisSelected AT %IX1425.7 : BOOL;	(*  ~ {LinkedWith:TIID^Device 1 (EtherCAT)^Rack 1 Slot 0 (EK1200)^Rack 1 Slot 15 (EL1008)^Channel 1^Input} *)
	.bARate1X AT %IX1426.0 : BOOL;	(*  ~ {LinkedWith:TIID^Device 1 (EtherCAT)^Rack 1 Slot 0 (EK1200)^Rack 1 Slot 15 (EL1008)^Channel 2^Input} *)
	.bARate10X AT %IX1426.1 : BOOL;	(*  ~ {LinkedWith:TIID^Device 1 (EtherCAT)^Rack 1 Slot 0 (EK1200)^Rack 1 Slot 15 (EL1008)^Channel 3^Input} *)
	.bARate100X AT %IX1426.2 : BOOL;	(*  ~ {LinkedWith:TIID^Device 1 (EtherCAT)^Rack 1 Slot 0 (EK1200)^Rack 1 Slot 15 (EL1008)^Channel 4^Input} *)
	.bWAAxisSelected AT %IX1426.3 : BOOL;	(*  ~ {LinkedWith:TIID^Device 1 (EtherCAT)^Rack 1 Slot 0 (EK1200)^Rack 1 Slot 15 (EL1008)^Channel 5^Input} *)
	.bXAAxisSelected AT %IX1426.4 : BOOL;	(*  ~ {LinkedWith:TIID^Device 1 (EtherCAT)^Rack 1 Slot 0 (EK1200)^Rack 1 Slot 15 (EL1008)^Channel 6^Input} *)
	.bYAAxisSelected AT %IX1426.5 : BOOL;	(*  ~ {LinkedWith:TIID^Device 1 (EtherCAT)^Rack 1 Slot 0 (EK1200)^Rack 1 Slot 15 (EL1008)^Channel 7^Input} *)
	.bZBAxisSelected AT %IX1426.6 : BOOL;	(*  ~ {LinkedWith:TIID^Device 1 (EtherCAT)^Box 20 (CU1128)^Rack 2 Slot 1 (EK1100)^Rack 2 Slot 3 (EL1008)^Channel 1^Input} *)
	.bBRate1X AT %IX1426.7 : BOOL;	(*  ~ {LinkedWith:TIID^Device 1 (EtherCAT)^Box 20 (CU1128)^Rack 2 Slot 1 (EK1100)^Rack 2 Slot 3 (EL1008)^Channel 2^Input} *)
	.bBRate10X AT %IX1427.0 : BOOL;	(*  ~ {LinkedWith:TIID^Device 1 (EtherCAT)^Box 20 (CU1128)^Rack 2 Slot 1 (EK1100)^Rack 2 Slot 3 (EL1008)^Channel 3^Input} *)
	.bBRate100X AT %IX1427.1 : BOOL;	(*  ~ {LinkedWith:TIID^Device 1 (EtherCAT)^Box 20 (CU1128)^Rack 2 Slot 1 (EK1100)^Rack 2 Slot 3 (EL1008)^Channel 4^Input} *)
	.bWBAxisSelected AT %IX1427.2 : BOOL;	(*  ~ {LinkedWith:TIID^Device 1 (EtherCAT)^Box 20 (CU1128)^Rack 2 Slot 1 (EK1100)^Rack 2 Slot 3 (EL1008)^Channel 5^Input} *)
	.bXBAxisSelected AT %IX1427.3 : BOOL;	(*  ~ {LinkedWith:TIID^Device 1 (EtherCAT)^Box 20 (CU1128)^Rack 2 Slot 1 (EK1100)^Rack 2 Slot 3 (EL1008)^Channel 6^Input} *)
	.bYBAxisSelected AT %IX1427.4 : BOOL;	(*  ~ {LinkedWith:TIID^Device 1 (EtherCAT)^Box 20 (CU1128)^Rack 2 Slot 1 (EK1100)^Rack 2 Slot 3 (EL1008)^Channel 7^Input} *)
	.bHighPressureMotorRunning AT %IX1427.5 : BOOL;	(*  ~ {LinkedWith:TIID^Device 1 (EtherCAT)^Box 20 (CU1128)^Rack 2 Slot 1 (EK1100)^Rack 2 Slot 4 (EL1008)^Channel 1^Input} *)
	.bTransferPumpMotorRunning AT %IX1427.6 : BOOL;	(*  ~ {LinkedWith:TIID^Device 1 (EtherCAT)^Box 20 (CU1128)^Rack 2 Slot 1 (EK1100)^Rack 2 Slot 4 (EL1008)^Channel 2^Input} *)
	.bChipConveyorMotorRunning AT %IX1427.7 : BOOL;	(*  ~ {LinkedWith:TIID^Device 1 (EtherCAT)^Box 20 (CU1128)^Rack 2 Slot 1 (EK1100)^Rack 2 Slot 4 (EL1008)^Channel 3^Input} *)
	.bHydraulicPowerUnitRunning AT %IX1428.0 : BOOL;	(*  ~ {LinkedWith:TIID^Device 1 (EtherCAT)^Box 20 (CU1128)^Rack 2 Slot 1 (EK1100)^Rack 2 Slot 4 (EL1008)^Channel 4^Input} *)
	.bMCC_V AT %IX1428.1 : BOOL;	(*  ~ {LinkedWith:TIID^Device 1 (EtherCAT)^Box 20 (CU1128)^Rack 2 Slot 1 (EK1100)^Rack 2 Slot 4 (EL1008)^Channel 5^Input} *)
	.bProx310 AT %IX1428.2 : BOOL;	(*  ~ {LinkedWith:TIID^Device 1 (EtherCAT)^Box 20 (CU1128)^Term 30 (CU1128-B)^Rack 3 (EP1008-0001)^Channel 1^Input} *)
	.bProx311 AT %IX1428.3 : BOOL;	(*  ~ {LinkedWith:TIID^Device 1 (EtherCAT)^Box 20 (CU1128)^Term 30 (CU1128-B)^Rack 3 (EP1008-0001)^Channel 2^Input} *)
	.bProx312 AT %IX1428.4 : BOOL;	(*  ~ {LinkedWith:TIID^Device 1 (EtherCAT)^Box 20 (CU1128)^Term 30 (CU1128-B)^Rack 3 (EP1008-0001)^Channel 3^Input} *)
	.bProx313 AT %IX1428.5 : BOOL;	(*  ~ {LinkedWith:TIID^Device 1 (EtherCAT)^Box 20 (CU1128)^Term 30 (CU1128-B)^Rack 3 (EP1008-0001)^Channel 4^Input} *)
	.bRack3Comm AT %IX1428.6 : BOOL;	(*  ~ {LinkedWith:TIID^Device 1 (EtherCAT)^Box 20 (CU1128)^Term 30 (CU1128-B)^Rack 3 (EP1008-0001)^WcState^WcState} *)
	.bProx410 AT %IX1428.7 : BOOL;	(*  ~ {LinkedWith:TIID^Device 1 (EtherCAT)^Box 20 (CU1128)^Term 30 (CU1128-B)^Rack 4 (EP1008-0001)^Channel 1^Input} *)
	.bProx411 AT %IX1429.0 : BOOL;	(*  ~ {LinkedWith:TIID^Device 1 (EtherCAT)^Box 20 (CU1128)^Term 30 (CU1128-B)^Rack 4 (EP1008-0001)^Channel 2^Input} *)
	.bProx412 AT %IX1429.1 : BOOL;	(*  ~ {LinkedWith:TIID^Device 1 (EtherCAT)^Box 20 (CU1128)^Term 30 (CU1128-B)^Rack 4 (EP1008-0001)^Channel 3^Input} *)
	.bProx413 AT %IX1429.2 : BOOL;	(*  ~ {LinkedWith:TIID^Device 1 (EtherCAT)^Box 20 (CU1128)^Term 30 (CU1128-B)^Rack 4 (EP1008-0001)^Channel 4^Input} *)
	.bProx414 AT %IX1429.3 : BOOL;	(*  ~ {LinkedWith:TIID^Device 1 (EtherCAT)^Box 20 (CU1128)^Term 30 (CU1128-B)^Rack 4 (EP1008-0001)^Channel 5^Input} *)
	.bProx415 AT %IX1429.4 : BOOL;	(*  ~ {LinkedWith:TIID^Device 1 (EtherCAT)^Box 20 (CU1128)^Term 30 (CU1128-B)^Rack 4 (EP1008-0001)^Channel 6^Input} *)
	.bRack4Comm AT %IX1429.5 : BOOL;	(*  ~ {LinkedWith:TIID^Device 1 (EtherCAT)^Box 20 (CU1128)^Term 30 (CU1128-B)^Rack 4 (EP1008-0001)^WcState^WcState} *)
	.bProx510 AT %IX1429.6 : BOOL;	(*  ~ {LinkedWith:TIID^Device 1 (EtherCAT)^Box 20 (CU1128)^Term 33 (CU1128-C)^Rack 5 (EP1008-0001)^Channel 1^Input} *)
	.bProx511 AT %IX1429.7 : BOOL;	(*  ~ {LinkedWith:TIID^Device 1 (EtherCAT)^Box 20 (CU1128)^Term 33 (CU1128-C)^Rack 5 (EP1008-0001)^Channel 2^Input} *)
	.bProx512 AT %IX1430.0 : BOOL;	(*  ~ {LinkedWith:TIID^Device 1 (EtherCAT)^Box 20 (CU1128)^Term 33 (CU1128-C)^Rack 5 (EP1008-0001)^Channel 3^Input} *)
	.bProx513 AT %IX1430.1 : BOOL;	(*  ~ {LinkedWith:TIID^Device 1 (EtherCAT)^Box 20 (CU1128)^Term 33 (CU1128-C)^Rack 5 (EP1008-0001)^Channel 4^Input} *)
	.bProx514 AT %IX1430.2 : BOOL;	(*  ~ {LinkedWith:TIID^Device 1 (EtherCAT)^Box 20 (CU1128)^Term 33 (CU1128-C)^Rack 5 (EP1008-0001)^Channel 5^Input} *)
	.bProx515 AT %IX1430.3 : BOOL;	(*  ~ {LinkedWith:TIID^Device 1 (EtherCAT)^Box 20 (CU1128)^Term 33 (CU1128-C)^Rack 5 (EP1008-0001)^Channel 6^Input} *)
	.bProx516 AT %IX1430.4 : BOOL;	(*  ~ {LinkedWith:TIID^Device 1 (EtherCAT)^Box 20 (CU1128)^Term 33 (CU1128-C)^Rack 5 (EP1008-0001)^Channel 7^Input} *)
	.bProx517 AT %IX1430.5 : BOOL;	(*  ~ {LinkedWith:TIID^Device 1 (EtherCAT)^Box 20 (CU1128)^Term 33 (CU1128-C)^Rack 5 (EP1008-0001)^Channel 8^Input} *)
	.bRack5Comm AT %IX1430.6 : BOOL;	(*  ~ {LinkedWith:TIID^Device 1 (EtherCAT)^Box 20 (CU1128)^Term 33 (CU1128-C)^Rack 5 (EP1008-0001)^WcState^WcState} *)
	.bProx610 AT %IX1430.7 : BOOL;	(*  ~ {LinkedWith:TIID^Device 1 (EtherCAT)^Box 20 (CU1128)^Term 33 (CU1128-C)^Rack 6 (EP1008-0001)^Channel 1^Input} *)
	.bProx611 AT %IX1431.0 : BOOL;	(*  ~ {LinkedWith:TIID^Device 1 (EtherCAT)^Box 20 (CU1128)^Term 33 (CU1128-C)^Rack 6 (EP1008-0001)^Channel 2^Input} *)
	.bProx612 AT %IX1431.1 : BOOL;	(*  ~ {LinkedWith:TIID^Device 1 (EtherCAT)^Box 20 (CU1128)^Term 33 (CU1128-C)^Rack 6 (EP1008-0001)^Channel 3^Input} *)
	.bProx613 AT %IX1431.2 : BOOL;	(*  ~ {LinkedWith:TIID^Device 1 (EtherCAT)^Box 20 (CU1128)^Term 33 (CU1128-C)^Rack 6 (EP1008-0001)^Channel 4^Input} *)
	.bProx614 AT %IX1431.3 : BOOL;	(*  ~ {LinkedWith:TIID^Device 1 (EtherCAT)^Box 20 (CU1128)^Term 33 (CU1128-C)^Rack 6 (EP1008-0001)^Channel 5^Input} *)
	.bProx615 AT %IX1431.4 : BOOL;	(*  ~ {LinkedWith:TIID^Device 1 (EtherCAT)^Box 20 (CU1128)^Term 33 (CU1128-C)^Rack 6 (EP1008-0001)^Channel 6^Input} *)
	.bPS616 AT %IX1431.5 : BOOL;	(*  ~ {LinkedWith:TIID^Device 1 (EtherCAT)^Box 20 (CU1128)^Term 33 (CU1128-C)^Rack 6 (EP1008-0001)^Channel 7^Input} *)
	.bPS617 AT %IX1431.6 : BOOL;	(*  ~ {LinkedWith:TIID^Device 1 (EtherCAT)^Box 20 (CU1128)^Term 33 (CU1128-C)^Rack 6 (EP1008-0001)^Channel 8^Input} *)
	.bRack6Comm AT %IX1431.7 : BOOL;	(*  ~ {LinkedWith:TIID^Device 1 (EtherCAT)^Box 20 (CU1128)^Term 33 (CU1128-C)^Rack 6 (EP1008-0001)^WcState^WcState} *)
	.bProx720 AT %IX1432.0 : BOOL;	(*  ~ {LinkedWith:TIID^Device 1 (EtherCAT)^Rack 7 (EP1008-0001)^Channel 1^Input} *)
	.bProx721 AT %IX1432.1 : BOOL;	(*  ~ {LinkedWith:TIID^Device 1 (EtherCAT)^Rack 7 (EP1008-0001)^Channel 2^Input} *)
	.bProx722 AT %IX1432.2 : BOOL;	(*  ~ {LinkedWith:TIID^Device 1 (EtherCAT)^Rack 7 (EP1008-0001)^Channel 3^Input} *)
	.bProx723 AT %IX1432.3 : BOOL;	(*  ~ {LinkedWith:TIID^Device 1 (EtherCAT)^Rack 7 (EP1008-0001)^Channel 4^Input} *)
	.bProx724 AT %IX1432.4 : BOOL;	(*  ~ {LinkedWith:TIID^Device 1 (EtherCAT)^Rack 7 (EP1008-0001)^Channel 5^Input} *)
	.bProx725 AT %IX1432.5 : BOOL;	(*  ~ {LinkedWith:TIID^Device 1 (EtherCAT)^Rack 7 (EP1008-0001)^Channel 6^Input} *)
	.bPS726 AT %IX1432.6 : BOOL;	(*  ~ {LinkedWith:TIID^Device 1 (EtherCAT)^Rack 7 (EP1008-0001)^Channel 7^Input} *)
	.bPS727 AT %IX1432.7 : BOOL;	(*  ~ {LinkedWith:TIID^Device 1 (EtherCAT)^Rack 7 (EP1008-0001)^Channel 8^Input} *)
	.bRack7Comm AT %IX1433.0 : BOOL;	(*  ~ {LinkedWith:TIID^Device 1 (EtherCAT)^Rack 7 (EP1008-0001)^WcState^WcState} *)
	.stReceivePanelA AT %IB74 : ST_PANEL_SEND;	(*  ~ {LinkedWith:TIID^Device 2 (EtherCAT Automation Protocol)^Panel A (Subscriber)^Panel_A_Send^Inputs^VarData} *)
	.nReceivePanelAQuality AT %IB738 : UINT;
	.nReceivePanelACycleIndex AT %IB740 : UINT;
	.nRequestPA AT %IB742 : WORD;	(*  ~ {LinkedWith:TIID^Device 2 (EtherCAT Automation Protocol)^Panel A (Subscriber)^Sub-Var 11^Inputs^VarData} *)
	.stReceivePanelB AT %IB744 : ST_PANEL_SEND;	(*  ~ {LinkedWith:TIID^Device 2 (EtherCAT Automation Protocol)^Panel B (Subscriber)^Panel_B_Send^Inputs^VarData} *)
	.nReceivePanelBQuality AT %IB1408 : UINT;
	.nReceivePanelBCycleIndex AT %IB1410 : UINT;
	.nRequestPB AT %IB1412 : WORD;	(*  ~ {LinkedWith:TIID^Device 2 (EtherCAT Automation Protocol)^Panel B (Subscriber)^Sub-Var 21^Inputs^VarData} *)
	.stCXPublish1 AT %QB4 : ST_CX_Publish1;	(*  ~ {LinkedWith:TIID^Device 2 (EtherCAT Automation Protocol)^CX_Publish 1 (Publisher)^Pub-Var 1^Outputs^VarData} *)
	.arrMachineInfo AT %QB1336 : ARRAY [1..20] OF STRING(30);	(*  ~ {LinkedWith:TIID^Device 2 (EtherCAT Automation Protocol)^Box 4 (Publisher)^Pub-Var Machine Info^Outputs^VarData} *)
	.stPartProgramSend AT %QB1956 : ST_PARTPROGRAM;	(*  ~ {LinkedWith:TIID^Device 2 (EtherCAT Automation Protocol)^Box 4 (Publisher)^Pub-Var Part program^Outputs^VarData} *)
	.nPubFrameState AT %IB1414 : UINT;
	.nVarCtrlMachineInfo AT %QB2256 : UINT;
	.nVarCtrlAutoDisplays AT %QB2258 : UINT;
	.nVarCtrlFaultMessages AT %QB2260 : UINT;
	.nVarCtrlPanelReceive AT %QB2262 : UINT;
	.nVarCtrlPartProgramSend AT %QB2264 : UINT;
	.nVarCtrlDemo AT %QB2266 : UINT;
	.stPB AT %IB1416 : ST_Demo_PBs;	(*  ~ {LinkedWith:TIID^Device 2 (EtherCAT Automation Protocol)^Panel A (Subscriber)^Sub-Var Demo^Inputs^VarData} *)
	.stPBB AT %IB1419 : ST_Demo_PBs;	(*  ~ {LinkedWith:TIID^Device 2 (EtherCAT Automation Protocol)^Panel B (Subscriber)^Sub-Var Demo^Inputs^VarData} *)
	.stLT AT %QB2268 : ST_Demo_Indicators;	(*  ~ {LinkedWith:TIID^Device 2 (EtherCAT Automation Protocol)^Box 4 (Publisher)^Pub-Var Demo^Outputs^VarData} *)
	.bAServoEnable AT %QX2273.0 : BOOL;	(*  ~ {LinkedWith:TIID^Device 1 (EtherCAT)^Rack 1 Slot 0 (EK1200)^Rack 1 Slot 5 (EL2809)^Channel 1^Output} *)
	.bBServoEnable AT %QX2273.1 : BOOL;	(*  ~ {LinkedWith:TIID^Device 1 (EtherCAT)^Rack 1 Slot 0 (EK1200)^Rack 1 Slot 5 (EL2809)^Channel 2^Output} *)
	.bUServoEnable AT %QX2273.2 : BOOL;	(*  ~ {LinkedWith:TIID^Device 1 (EtherCAT)^Rack 1 Slot 0 (EK1200)^Rack 1 Slot 5 (EL2809)^Channel 3^Output} *)
	.bMCC_S AT %QX2273.3 : BOOL;	(*  ~ {LinkedWith:TIID^Device 1 (EtherCAT)^Rack 1 Slot 0 (EK1200)^Rack 1 Slot 5 (EL2809)^Channel 4^Output} *)
	.bWayLubePump AT %QX2273.4 : BOOL;	(*  ~ {LinkedWith:TIID^Device 1 (EtherCAT)^Rack 1 Slot 0 (EK1200)^Rack 1 Slot 5 (EL2809)^Channel 5^Output} *)
	.bACoolantSolenoid AT %QX2273.5 : BOOL;	(*  ~ {LinkedWith:TIID^Device 1 (EtherCAT)^Rack 1 Slot 0 (EK1200)^Rack 1 Slot 5 (EL2809)^Channel 6^Output} *)
	.bBCoolantSolenoid AT %QX2273.6 : BOOL;	(*  ~ {LinkedWith:TIID^Device 1 (EtherCAT)^Rack 1 Slot 0 (EK1200)^Rack 1 Slot 5 (EL2809)^Channel 7^Output} *)
	.bConveyorFWDReq AT %QX2273.7 : BOOL;	(*  ~ {LinkedWith:TIID^Device 1 (EtherCAT)^Rack 1 Slot 0 (EK1200)^Rack 1 Slot 5 (EL2809)^Channel 8^Output} *)
	.bHPCoolantStart_A AT %QX2274.0 : BOOL;	(*  ~ {LinkedWith:TIID^Device 1 (EtherCAT)^Rack 1 Slot 0 (EK1200)^Rack 1 Slot 5 (EL2809)^Channel 9^Output} *)
	.bHPCoolantStart_B AT %QX2274.1 : BOOL;	(*  ~ {LinkedWith:TIID^Device 1 (EtherCAT)^Rack 1 Slot 0 (EK1200)^Rack 1 Slot 5 (EL2809)^Channel 10^Output} *)
	.bTransferDown AT %QX2274.2 : BOOL;	(*  ~ {LinkedWith:TIID^Device 1 (EtherCAT)^Rack 1 Slot 0 (EK1200)^Rack 1 Slot 5 (EL2809)^Channel 11^Output} *)
	.bTransferUp AT %QX2274.3 : BOOL;	(*  ~ {LinkedWith:TIID^Device 1 (EtherCAT)^Rack 1 Slot 0 (EK1200)^Rack 1 Slot 5 (EL2809)^Channel 12^Output} *)
	.bATailstockColletUnclamp AT %QX2274.4 : BOOL;	(*  ~ {LinkedWith:TIID^Device 1 (EtherCAT)^Rack 1 Slot 0 (EK1200)^Rack 1 Slot 5 (EL2809)^Channel 13^Output} *)
	.bATailstockColletClamp AT %QX2274.5 : BOOL;	(*  ~ {LinkedWith:TIID^Device 1 (EtherCAT)^Rack 1 Slot 0 (EK1200)^Rack 1 Slot 5 (EL2809)^Channel 14^Output} *)
	.bBTailstockColletUnclamp AT %QX2274.6 : BOOL;	(*  ~ {LinkedWith:TIID^Device 1 (EtherCAT)^Rack 1 Slot 0 (EK1200)^Rack 1 Slot 5 (EL2809)^Channel 15^Output} *)
	.bBTailstockColletClamp AT %QX2274.7 : BOOL;	(*  ~ {LinkedWith:TIID^Device 1 (EtherCAT)^Rack 1 Slot 0 (EK1200)^Rack 1 Slot 5 (EL2809)^Channel 16^Output} *)
	.bAEjectorsRetract AT %QX2275.0 : BOOL;	(*  ~ {LinkedWith:TIID^Device 1 (EtherCAT)^Rack 1 Slot 0 (EK1200)^Rack 1 Slot 6 (EL2809)^Channel 1^Output} *)
	.bAEjectorsAdvance AT %QX2275.1 : BOOL;	(*  ~ {LinkedWith:TIID^Device 1 (EtherCAT)^Rack 1 Slot 0 (EK1200)^Rack 1 Slot 6 (EL2809)^Channel 2^Output} *)
	.bBEjectorsRetract AT %QX2275.2 : BOOL;	(*  ~ {LinkedWith:TIID^Device 1 (EtherCAT)^Rack 1 Slot 0 (EK1200)^Rack 1 Slot 6 (EL2809)^Channel 3^Output} *)
	.bBEjectorsAdvance AT %QX2275.3 : BOOL;	(*  ~ {LinkedWith:TIID^Device 1 (EtherCAT)^Rack 1 Slot 0 (EK1200)^Rack 1 Slot 6 (EL2809)^Channel 4^Output} *)
	.bChipConveyorFWD AT %QX2275.4 : BOOL;	(*  ~ {LinkedWith:TIID^Device 1 (EtherCAT)^Rack 1 Slot 0 (EK1200)^Rack 1 Slot 6 (EL2809)^Channel 9^Output} *)
	.bLT2 AT %QX2275.5 : BOOL;	(*  ~ {LinkedWith:TIID^Device 1 (EtherCAT)^Rack 1 Slot 0 (EK1200)^Rack 1 Slot 6 (EL2809)^Channel 11^Output} *)
	.bLT3 AT %QX2275.6 : BOOL;	(*  ~ {LinkedWith:TIID^Device 1 (EtherCAT)^Rack 1 Slot 0 (EK1200)^Rack 1 Slot 6 (EL2809)^Channel 12^Output} *)
	.bLT4 AT %QX2275.7 : BOOL;	(*  ~ {LinkedWith:TIID^Device 1 (EtherCAT)^Rack 1 Slot 0 (EK1200)^Rack 1 Slot 6 (EL2809)^Channel 13^Output} *)
	.bLT5 AT %QX2276.0 : BOOL;	(*  ~ {LinkedWith:TIID^Device 1 (EtherCAT)^Rack 1 Slot 0 (EK1200)^Rack 1 Slot 6 (EL2809)^Channel 14^Output} *)
	.bLT6 AT %QX2276.1 : BOOL;	(*  ~ {LinkedWith:TIID^Device 1 (EtherCAT)^Box 20 (CU1128)^Rack 2 Slot 1 (EK1100)^Rack 2 Slot 6 (EL2008)^Channel 1^Output} *)
	.bHighPressureMotorOn AT %QX2276.2 : BOOL;	(*  ~ {LinkedWith:TIID^Device 1 (EtherCAT)^Box 20 (CU1128)^Rack 2 Slot 1 (EK1100)^Rack 2 Slot 6 (EL2008)^Channel 2^Output} *)
	.bTransferPumpOn AT %QX2276.3 : BOOL;	(*  ~ {LinkedWith:TIID^Device 1 (EtherCAT)^Box 20 (CU1128)^Rack 2 Slot 1 (EK1100)^Rack 2 Slot 6 (EL2008)^Channel 3^Output} *)
	.bHydraulicUnitOn AT %QX2276.4 : BOOL;	(*  ~ {LinkedWith:TIID^Device 1 (EtherCAT)^Box 20 (CU1128)^Rack 2 Slot 1 (EK1100)^Rack 2 Slot 6 (EL2008)^Channel 5^Output} *)
	.bChipConveyorOn AT %QX2276.5 : BOOL;	(*  ~ {LinkedWith:TIID^Device 1 (EtherCAT)^Box 20 (CU1128)^Rack 2 Slot 1 (EK1100)^Rack 2 Slot 6 (EL2008)^Channel 4^Output} *)
	.bVFD_A_Enable AT %QX2276.6 : BOOL;	(*  ~ {LinkedWith:TIID^Device 1 (EtherCAT)^Box 20 (CU1128)^Rack 2 Slot 1 (EK1100)^Rack 2 Slot 7 (EL2008)^Channel 1^Output} *)
	.bVFD_B_Enable AT %QX2276.7 : BOOL;	(*  ~ {LinkedWith:TIID^Device 1 (EtherCAT)^Box 20 (CU1128)^Rack 2 Slot 1 (EK1100)^Rack 2 Slot 7 (EL2008)^Channel 2^Output} *)
END_VAR

(* Data type *)
TYPE AutoCycleStates :
(
	AC_Init:=0,
	AC_TransferParts,
	AC_Clamp,
	AC_ReturnTransfer,
	AC_CoolantOn,
	AC_SpindleOn,
	AC_Drill,
	AC_Retract,
	AC_SpindleOff,
	AC_CoolantOff,
	AC_Unclamp,
	AC_Finish,
	AC_CellRunoutFinish,
	AC_DrillReturn
);
END_TYPE

(* Data type *)
TYPE AutoModeStates :
(
	AM_NotInCycle:=0,
	AM_RetractZAxis,
	AM_InCycle,
	AM_GotoManualMode
);
END_TYPE

(* Data type *)
TYPE Ke_Energy :
STRUCT
	fEnergy:LREAL:=0.0;
	sUnits:STRING(3):='kWh';
END_STRUCT
END_TYPE

(* Data type *)
TYPE Ke_ErrorCodev2 :
(
	Er_NoError:=0,
	Er_MotorStarterFailed,
	Er_ServoWarning,
	Er_ServoFault,
	Er_InvalidParameters,
	Er_DrillReturn,
	Er_InvalidToolDiameter,
	Er_InvalidIPM,
	Er_InvalidIPR,
	Er_InvalidRPM,
	Er_InvalidSFM,
	Er_InvalidRatio,
	Er_InvalidOverride,
	Er_InvalidIPAddress,
	Er_UpToSpeedTimeout,
	Er_DriveNotReady,
	Er_DriveFaulted,
	Er_DriveWarning,
	Er_DriveComm,
	Er_NoJogRate,
	Er_NoRapidRate
);
END_TYPE

(* Would like to eleminate this Data Type *)

(* Data type *)
TYPE Ke_OperationTime :
STRUCT
	nYears:UINT:=0;
	nDays:UINT:=0;
	nHours:UINT:=0;
	nMinutes:UINT:=0;
	nSeconds:UINT:=0;
END_STRUCT
END_TYPE

(* Data type *)
TYPE Ke_VFDInfo :
STRUCT
	bDataValid:BOOL;
	nStatusWord:WORD;
	nControlWord:WORD;
	nReferenceSpeed:UINT;
	nActualSpeed:UINT;
	fFrequencyReference:LREAL;
	fFrequencyOut:LREAL;
	fFrequencyMin:LREAL;
	fFrequencyMax:LREAL;
	nFrequencyScale:USINT;
	nMotorSpeed:INT;
	nMotorNominalSpeed:INT;
	fMotorNominalFrequency:LREAL;
	fMotorVoltage:LREAL;
	fMotorNominalVoltage:LREAL;
	fMotorCurrent:LREAL;
	fMotorNominalCurrent:LREAL;
	nCurrentScale:UINT;
	fMotorCurrentLimit:LREAL;
	fMotorTorque:LREAL;
	fMotorPower:LREAL;
	fAccelerationTime:LREAL;
	fDecelerationTime:LREAL;
	fRampTimeScale:LREAL;
	nPolePairNumber:UINT;
	nDCLinkVoltage:UINT;
	nActiveFault:USINT;
	stDayCounter:Ke_OperationTime;
	stDayCounterResettable:Ke_OperationTime;
	stEnergyCounter:Ke_Energy;
	stEnergyCounterResettable:Ke_Energy;
	arrFaultHistory:ARRAY[1..16] OF WORD;
END_STRUCT
END_TYPE

(* Data type *)
TYPE Ke_VFDState :
(
	VFD_NotReady:=0,
	VFD_Ready,
	VFD_Run,
	VFD_Fault,
	VFD_OpDayReset,
	VFD_EnergyReset,
	VFD_Run_Setup,
	VFD_Run_Request,
	VFD_Run_AtSpeed,
	VFD_Run_Override,
	VFD_Run_Stop
);
END_TYPE

(* Data type *)
TYPE ManualModeStates :
(
	MM_Nothing:=0,
	MM_JogForward:=1,
	MM_JogReverse,
	MM_IncrForward,
	MM_IncrReverse,
	MM_SetZAZero,
	MM_SetZBZero,
	MM_MoveZAToZero,
	MM_MoveZBToZero,
	MM_CounterRotationJog,
	MM_Setup,
	MM_SetupModeAWSpindle,
	MM_SetupModeBWSpindle,
	MM_GotoAutomaticMode,
	MM_CoolantOn,
	MM_CoolantOff,
	MM_Calculate,
	MM_MakeOverrideCurrent,
	MM_MakeCalculatedCurrent,
	MM_ClampPart,
	MM_UnclampPart,
	MM_MPGToggle,
	MM_HydraulicUnitStart,
	MM_HydraulicUnitStop,
	MM_HomeZAxis,
	MM_HomeAutomation,
	MM_XMPG,
	MM_YMPG,
	MM_ZMPG,
	MM_WMPG
);
END_TYPE

(* Data type *)
TYPE ModeErrors :
(
	Er_NoModeError:=0,
	Er_CoolantOff:=1,
	Er_CleanTankLow,
	Er_CoolantOverflow,
	Er_HPPumpOff,
	Er_AMClampTimeout,
	Er_AMCoolantTimeout,
	Er_VFDUpToSpeedTimeout,
	Er_MMCoolantStartTimeout,
	Er_MMCoolantValveStopTimeout,
	Er_AMUnclampTimeout,
	Er_MPG_A_Active,
	Er_MPG_B_Active,
	Er_HydraulicPSOff,
	Er_XAxisNotHomed,
	Er_TransferNotAtLoad,
	Er_ZAAxisNotHomed,
	Er_WAAxisNotHomed,
	Er_WANotRetracted,
	Er_ACulletNotUnclamped,
	Er_AEjectorsNotRetracted,
	Er_ZBAxisNotHomed,
	Er_WBAxisNotHomed,
	Er_WBNotRetracted,
	Er_BCulletNotUnclamped,
	Er_BEjectorsNotRetracted,
	Er_EMNoAuto,
	Er_SetupError,
	Er_PartNotUnclamped,
	Er_PartUnclamped,
	Er_LoadPartMissing,
	Er_UnloadPartPresent,
	Er_ZAHomeError,
	Er_ZBHomeError,
	Er_ZAMoveError,
	Er_ZBMoveError,
	Er_HomeTimeout,
	Er_TryingToLeaveAutoInCycle,
	Er_TransferSolError,
	Er_SideAColletSolError,
	Er_SideBColletSolError,
	Er_SideAEjectorsSolError,
	Er_SideBEjectorsSolError,
	Er_MaxCyclesReached
);
END_TYPE

(* Data type *)
TYPE ST_CX_Publish1 :
	(******* Replace Auto Display, Fault String, and panel Receive Structures ****************)
STRUCT
	(* The structure of Arrays are Published by the CX program.  We must use this definition to decrypt  them in the translate PRG
		The arrays should be at least 25%  greater than what is used, So we do not have to re-define the structure and 
		re-establish the communication connections *)
	arrUDINTIGER: ARRAY[1..50] OF UDINT := 0;
	arrLREAL: ARRAY[1..50] OF LREAL := 0.0;
	arrSTRING50 : ARRAY[1..12] OF STRING (52) := 12('');
	arrBOOL: ARRAY[1..96] OF BOOL:= FALSE;

END_STRUCT
END_TYPE

(* Data type *)
TYPE ST_Demo_Indicators :
STRUCT
	LT1A:BOOL;
	LT2A:BOOL;
	LT1B:BOOL;
	LT2B:BOOL;
	LTCom:BOOL;
END_STRUCT
END_TYPE

(* Data type *)
TYPE ST_Demo_PBs :
STRUCT
	bPB1:BOOL;
	bPB2:BOOL;
	bPB3:BOOL;
END_STRUCT
END_TYPE

(* Data type *)
TYPE ST_PANEL_SEND :
STRUCT
	(* The structure of  Arrays sent to the CX program are encripted in the Translate PRG.  The CX must use this definition to decript them it's program
	    The arrays should be at least 25%  greater than what is used, So we do not have to re-define the structure and re-establish the communication connections *)
	arrUDINTIGER: ARRAY[1..20] OF UDINT := 0;
	arrLREAL: ARRAY[1..32] OF LREAL := 0.0;
	arrBOOL: ARRAY[1..96] OF BOOL:= FALSE;
	arrTEXTSTRING: ARRAY[1..8] OF STRING (28) := 8('');

END_STRUCT
END_TYPE

(* Data type *)
TYPE ST_PARTPROGRAM :
	(* The structure of Arrays are defined in the CX program.  We must use this definition to decript them in the translate PRG
		The arrays should be at least 25%  greater than what is used, So we do not have to re-define the structure and 
		re-establish the communication connections *)
STRUCT
	(*  This structure are variables of the Part Program to be displayed when on the Part Program Screen *)
	arrLREAL : ARRAY[1..18] OF LREAL := 0.0;
	arrSTRING : ARRAY[1..4] OF STRING(30) := 3('');
	arrBOOL: ARRAY[1..32] OF BOOL:= FALSE;

END_STRUCT
END_TYPE

(* POU Programs/MAIN, ST *)
PROGRAM MAIN
VAR
	fbMCC_STon : TON;				(* Delay Timer for Servo Power *)

	(*	Manual Mode Helper Variables *)
	nManualModeState: ManualModeStates := MM_Nothing;
	fbSetupModeATimer: TON;
	fbSetupModeBTimer: TON;
	fbSoftStartTimer: TON;
	fbSoftStartTimer2: TON;
	fbCleanTankLevelDelay: TON;						(* Clean Tank Float Switch must be on for 2 seconds *)
	fbMachineModeChangeRTrig : R_TRIG;
	bAutoModeRequest : BOOL := FALSE;
	bManModeRequest : BOOL := FALSE;
	bCoolantSolenoidControl : BOOL := FALSE;			(* Used to Turn On the High Pressure Coolant Solenoids *)
	bStoppingSetup: BOOL := FALSE;
	fbStoppingSetupTON: TON;
	nHomeAutomationStep: INT;						(* Counter for MM_HomeAutomation Steps *)
	fbHomeTimer:TON;								(* Timer used in Homing Automation *)

	(*	Hydraulic Power Unit Control Variables *)
	fbHydraulicPowerUnitMotorControl: FB_MotorStarter;
	bHydraulicPowerUnitMotorControl: BOOL := FALSE;
	bHydraulicPowerUnitMotorControlError: BOOL := FALSE;

	(*	Transfer Pump Control Variables *)
	fbTransferPumpMotorControl: FB_MotorStarter;
	bTransferPumpMotorControl: BOOL := FALSE;
	bTransferPumpMotorControlError: BOOL := FALSE;

	(*	High Pressure Motor Control Variables *)
	fbHighPressureMotorControl: FB_MotorStarter;
	bHighPressureMotorControl: BOOL := FALSE;
	bHighPressureMotorControlError: BOOL := FALSE;

	(*	Chip Conveyor Control Variables *)
	fbChipConveyorMotorControl: FB_MotorStarter;
	bChipConveyorMotorControl: BOOL := FALSE;
	bChipConveyorMotorControlError: BOOL := FALSE;

	(* Auto Cycle Variables *)
	tLastCycleTime: TIME := t#0s;
	fbCycleTimer: TON;
	bCycleTimer: BOOL;
	fbFaultLightBlink: TON;
	bFaultLightBlink: BOOL := FALSE;

	(*	Cycle Start Control Variables *)
	fbCycleStartControl: FB_CycleStart;
	bCycleStartControlHold: BOOL := FALSE;
	bCycleStartControlReset: BOOL := FALSE;
	bCycleStartControlEnable: BOOL := FALSE;

	bCoolantTimer: BOOL := FALSE;
	tCoolantTime: TIME := t#0s;
	fbCoolantTimer: TON;
	tCycleDelayTime: TIME := t#0s;
	fbPS1DelayTON: TON;							(* Delay of PS1- Side A coolant ON *)
	fbPS2DelayTON: TON;							(* Delay of PS1- Side B coolant ON *)
	fbUpToSpeedATON: TON;						(* Delay of Side A VFD's Up to Speed Bits *)
	fbUpToSpeedBTON: TON;						(* Delay of Side B VFD's Up to Speed Bits *)
	fbDwellTimeTON: TON;						(* Drill cycle Dwell Timer *)
	tDwellTime: TIME := t#0s;						(* Drill Cycle Dwell Time *)
	bDwellTime: BOOL := FALSE;					(* Drill Cycle Dwell Timer Trigger *)
	nDrillStep : INT :=0;							(* State counter for AC_Drill Step *)

	bCycleWatchdogTimer: BOOL := FALSE;			(* In Cycle Watchdog Timer Trigger *)
	tCycleWatchdogTime: TIME := t#0ms;				(* In Cycle Watchgod Timer - Time *)
	fbCycleWatchdogTimer : TON;					(*In Cycle Watchdog Timer *)
	bUnclampDelayTimer : BOOL := FALSE;			(* Trigger the dealy timer in the Unclamp Cycle *)
	fbUnclampDelayTON : TON;					(* Unclamp Cycle Delay Timer *)

	nVFDControlRPM: UINT := 0;					(* Spindle RPM Request Converted into Intiger*)
	fbVFD_AStarting: R_TRIG;						(* VFD's for Side A Start Trigger *)
	fbVFD_AHealthyTON: TON;						(* Delay theSide A VFD Healthy signal *)
	fbVFD_BStarting: R_TRIG;						(* VFD's for Side A Start Trigger *)
	fbVFD_BHealthyTON: TON;						(* Delay theSide B VFD Healthy signal *)
	fbVFD_A_EnableTON: TON;					(* Delay of the Side A VFD Enable Signal for Interanal Reset *)
	fbVFD_B_EnableTON: TON;					(* Delay of the Side B VFD Enable Signal for Interanal Reset *)
	fbAResetInternalTrig: R_TRIG;					(* Trigger and internal Reset based on Side A VFD's Status *)
	fbBResetInternalTrig: R_TRIG;					(* Trigger and internal Reset based on Side B VFD's Status *)

	nRPMScaleMax: UDINT := 2500;			(* Max scale set in the Red Lion IFMA modules *)
	bFaultLight: BOOL := FALSE;			(* Panel Fault Lights *)
	bTowerFaultLight: BOOL := FALSE;		(* Tower Red Fault Light*)
	bTowerNotInCycle: BOOL := FALSE;		(* Tower Amber Light *)
	bTowerInCycle: BOOL := FALSE;			(* Tower Green Light *)
	bSetupModeA: BOOL := FALSE;			(*Setup Mode Incudes Side A*)
	nSetupModeAStep: INT := 0;			(* Step Counter for Side A Setup *)
	bSetupModeB: BOOL := FALSE;			(*Setup Mode Includes Side B *)
	nSetupModeBStep: INT := 0;			(* Step Counter for Side B Setup *)
	nDrillReturnCount: INT := 0;				(* Drill Return Counter*)
	fbPB1AConfirmRTrig: R_TRIG;			(* Rising Trigger of Side A Confirm Button *)
	fbPB1BConfirmRTrig: R_TRIG;			(* Rising Trigger of Side B Confirm Button *)
	nCountA: INT := 0;		(*Counter for Test purposes *)
	nCountB: INT := 0;		(*Counter for test purposes *)
	fbVFD_ADataValid: TON;		(* Valid Data from Side A Drives *)
	fbVFD_BDataValid: TON;		(* Valid Data from Side A Drives *)

END_VAR
IF stUAxis.NcToPlc.StateDWord.1 AND
	(stWAAxis.NcToPlc.StateDWord.1 OR NOT bSideAEnabled) AND
	(stWBAxis.NcToPlc.StateDWord.1 OR NOT bSideBEnabled)
THEN
	bWandUAxisHomed := TRUE;
ELSE
	bWandUAxisHomed := FALSE;
END_IF

(* Run the Way Lube when the MCR is On *)
bWayLubePump:= bMCR;

(* Delay the Servo Power after the MCR comes on *)
fbMCC_STon(IN:=bMCR, PT:= t#2s);
bMCC_S := fbMCC_STon.Q;
bMCC_SConfirm;		(* Display Feedback *)

(* When the MCC_S comes in then turn on the Hard Enables *)
bUServoEnable := bMCC_SConfirm;
IF bSideAEnabled THEN
	bAServoEnable := bMCC_SConfirm;
ELSE
	bAServoEnable := FALSE;
END_IF
IF bSideBEnabled THEN
	bBServoEnable := bMCC_SConfirm;
ELSE
	bBServoEnable := FALSE;
END_IF


(*			POWER ON			*)
IF bMCR THEN

	(* VFD Contactor on *)
	IF bMCC_V THEN
		(* Side A Spindle VFD's Enable *)
		IF bSideAEnabled THEN
			IF fbVFD_AHealthyTON.Q AND fbVFD_ADataValid.Q THEN
				bVFD_A_Enable:=TRUE;
			ELSE
				bVFD_A_Enable:=FALSE;
			END_IF
		ELSE
			bVFD_A_Enable:=FALSE;
		END_IF

		(* Side B Spindle VFD's Enable *)
		IF bSideBEnabled THEN
			IF fbVFD_BHealthyTON.Q AND fbVFD_BDataValid.Q THEN
				bVFD_B_Enable:=TRUE;
			ELSE
				bVFD_B_Enable:=FALSE;
			END_IF
		ELSE
			bVFD_B_Enable:=FALSE;
		END_IF

	END_IF

	(*****  CHANGE MANUAL AND AUTO MODES ******)
	(* Check Conditions before going into Auto *)
	(* Check Warnings and Faults *)
	IF NOT bMachineMode AND fbMachineModeChangeRTrig.Q AND NOT bMachineWarning AND NOT bMachineFault THEN
		(* Check MPG A Off *)
		IF bMPGAOn THEN
			nModeError:=Er_MPG_A_Active;
		(* Check MPG B Off *)
		ELSIF bMPGBOn THEN
			nModeError:=Er_MPG_B_Active;
		(* Check Hydraulic Pressure Switch *)
		ELSIF NOT bHydraulicSystemPressure  THEN
			nModeError:=Er_HydraulicPSOff;
		(* Check Coolant High Pressure Pump On *)
		ELSIF NOT bHighPressureMotorRunning THEN
			nModeError:=Er_HPPumpOff;
		(* Check Homing of Transfer *)
		ELSIF NOT stUAxis.NcToPlc.StateDWord.1 THEN
			nModeError:=Er_XAxisNotHomed;
		(*Check Transfer Position *)
		ELSIF NOT bTransferAtLoadIndicator THEN
			nModeError:=Er_TransferNotAtLoad;
		(*Check Homing of ZA Axis *)
		ELSIF bSideAEnabled AND NOT stZAAxis.NcToPlc.StateDWord.1 THEN
			nModeError:=Er_ZAAxisNotHomed;
		(*Check Homing of WA Axis *)
		ELSIF bSideAEnabled AND NOT stWAAxis.NcToPlc.StateDWord.1 THEN
			nModeError:=Er_WAAxisNotHomed;
		(*Check Position of WA Tailstock *)
		ELSIF bSideAEnabled AND stWAAxis.NcToPlc.ActPos < (fWAxisTransferPosition-0.2)   THEN
			nModeError:=Er_WANotRetracted;
		(* Check Side A Cullets Unclamped *)
		ELSIF bSideAEnabled AND NOT bPS616 THEN
			nModeError:=Er_ACulletNotUnclamped;
		(* Check Side A Ejectors Retracted *)
		ELSIF bSideAEnabled AND NOT (nAEjectorRetractedState=7 AND nAEjectorAdvancedState=7) THEN
			nModeError:=Er_AEjectorsNotRetracted;
		(*Check Homing of ZB Axis *)
		ELSIF bSideBEnabled AND NOT stZBAxis.NcToPlc.StateDWord.1 THEN
			nModeError:=Er_ZBAxisNotHomed;
		(*Check Homing of WB Axis *)
		ELSIF bSideBEnabled AND NOT stWBAxis.NcToPlc.StateDWord.1 THEN
			nModeError:=Er_WBAxisNotHomed;
		(*Check Position of WB Tailstock *)
		ELSIF bSideBEnabled AND stWBAxis.NcToPlc.ActPos < (fWAxisTransferPosition-0.2)   THEN
			nModeError:=Er_WBNotRetracted;
		(* Check Side B Cullets Unclamped *)
		ELSIF bSideBEnabled AND NOT bPS726 THEN
			nModeError:=Er_BCulletNotUnclamped;
		(* Check Side A Ejectors Retracted *)
		ELSIF bSideBEnabled AND NOT (nBEjectorRetractedState=7 AND nBEjectorAdvancedState=7) THEN
			nModeError:=Er_BEjectorsNotRetracted;
		(* Passed Checks - Enter Auto Mode *)
		ELSE
			bMachineMode := TRUE;
		END_IF
	(* Check Conditions before going into Manual *)
	ELSIF bMachineMode AND fbMachineModeChangeRTrig.Q THEN
		IF NOT bInCycle THEN
			bMachineMode := FALSE;
		ELSE
			nModeError:=Er_TryingToLeaveAutoInCycle;
		END_IF
	END_IF


	(*		MANUAL MODE FUNCTIONS 		*)
	IF NOT bMachineMode THEN
		(*Turn Off all Auoto Mode bits *)
		bAutoTransferPartsToDrill:=FALSE;
		bAutoTransferDownAndLoad := FALSE;
		bLoadPartsConfirmed:= FALSE;
		bUnloadPartsConfirmed:=FALSE;
		bInCycle:=FALSE;
		bCycleTimer:=FALSE;
		nAutoModeState:=AM_NotInCycle;
		nAutoCycleStep:=AC_Init;
		bCellRunoutRequest:=FALSE;
		bCycleWatchdogTimer := FALSE;
		bAutoClampAStart:=FALSE;
		bAutoClampBStart:=FALSE;
		bAutoUnclampAStart:=FALSE;
		bAutoUnclampBStart:=FALSE;
		bCoolantTimer:= FALSE;
		nAC_UnclampStep := 0;

		(* Reset the Counters when the PB's are pressed *)
		IF bResetCycleCounterPB THEN
			nCyclesComplete:=0;
		ELSIF bResetTotalCountPB THEN
			nPartsCompleteTotal:=0;
		ELSIF bResetA1CountPB THEN
			nPartsCompleteA1:=0;
		ELSIF bResetA2CountPB THEN
			nPartsCompleteA2:=0;
		ELSIF bResetA3CountPB THEN
			nPartsCompleteA3:=0;
		ELSIF bResetB1CountPB THEN
			nPartsCompleteB1:=0;
		ELSIF bResetB2CountPB THEN
			nPartsCompleteB2:=0;
		ELSIF bResetB3CountPB THEN
			nPartsCompleteB3:=0;

		END_IF

		CASE nManualModeState OF
		MM_Nothing:

			IF bStopHydraulicPB THEN
				bHydraulicPowerUnitMotorControl:=FALSE;
			ELSIF bCoolantStopPB THEN
				nManualModeState:=MM_CoolantOff;
			ELSIF bMachineFault THEN
				(* Coolant Related Faults *)
				IF nActiveFaults[1].2=1			(* High Pressure Pump MS Failure *)
					OR nActiveFaults[1].3=1	(* Transfer Pump MS Failure *)
					OR nActiveFaults[1].5=1	(* Low Float Switch *)
					OR nActiveFaults[1].6=1	(* High Coolant Temp Fault *)
					OR bCoolantStopPB		(* Allow Operator to shut off Coolant sytem *)
				 THEN
					nManualModeState:=MM_CoolantOff;
				END_IF
			ELSIF bStartHydraulicPB AND NOT bHydraulicPowerUnitMotorControlError THEN
				bHydraulicPowerUnitMotorControl:=TRUE;
			ELSIF bCoolantStartPB THEN
				nManualModeState:=MM_CoolantOn;
			ELSIF bEnterSetupPB_A THEN
				nManualModeState:=MM_Setup;
			ELSIF bEnterSetupPB_B THEN
				nManualModeState:=MM_Setup;
			ELSIF bSetZeroPositionPB_A THEN
				nManualModeState:=MM_SetZAZero;
			ELSIF bSetZeroPositionPB_B THEN
				nManualModeState:=MM_SetZBZero;
			ELSIF bMoveToZeroPositionPB_A THEN
				nManualModeState:=MM_MoveZAToZero;
			ELSIF bMoveToZeroPositionPB_B THEN
				nManualModeState:=MM_MoveZBToZero;
			ELSIF bHomeAutomationPB THEN
				IF bMPGAOn THEN
					nModeError:=Er_MPG_A_Active;
				ELSIF bMPGBOn THEN
					nModeError:=Er_MPG_B_Active;
				ELSE
					nHomeAutomationStep:=0;
					nManualModeState:=MM_HomeAutomation;
				END_IF
			END_IF

		MM_Setup:
			IF bEnterSetupPB_A THEN
				bSetupModeA:=TRUE;
			END_IF
			IF bEnterSetupPB_B THEN
				bSetupModeB:=TRUE;
			END_IF

